LIN {X 0,Y 197.752,Z 444.521,A -85,B 0,C 180,E1 -22110.162,E2 -22110.162} C_VEL
LIN {X 0,Y 204.908,Z 442.853,A -85,B 0,C 180,E1 -22106.718,E2 -22106.718} C_VEL
LIN {X 0,Y 212.782,Z 440.264,A -85,B 0,C 180,E1 -22103.522,E2 -22103.522} C_VEL
LIN {X 0,Y 223.864,Z 435.745,A -85,B 0,C 180,E1 -22099.941,E2 -22099.941} C_VEL
LIN {X 0,Y 233.532,Z 431.085,A -85,B 0,C 180,E1 -22097.381,E2 -22097.381} C_VEL
LIN {X 0,Y 236.072,Z 429.745,A -85,B 0,C 180,E1 -22096.787,E2 -22096.787} C_VEL
LIN {X 0,Y 232.311,Z 432.152,A -85,B 0,C 180,E1 -22095.84,E2 -22095.84} C_VEL
LIN {X 0,Y 218.81,Z 440.079,A -85,B 0,C 180,E1 -22092.416,E2 -22092.416} C_VEL
LIN {X 0,Y 207.624,Z 445.92,A -85,B 0,C 180,E1 -22088.772,E2 -22088.772} C_VEL
LIN {X 0,Y 198.004,Z 450.413,A -85,B 0,C 180,E1 -22084.605,E2 -22084.605} C_VEL
LIN {X 0,Y 191.543,Z 453.093,A -85,B 0,C 180,E1 -22080.909,E2 -22080.909} C_VEL
LIN {X 0,Y 186.17,Z 454.953,A -85,B 0,C 180,E1 -22076.937,E2 -22076.937} C_VEL
LIN {X 0,Y 180.265,Z 456.156,A -85,B 0,C 180,E1 -22070.662,E2 -22070.662} C_VEL
LIN {X 0,Y 178.735,Z 456.196,A -85,B 0,C 180,E1 -22067.89,E2 -22067.89} C_VEL
LIN {X 0,Y 177.023,Z 461.145,A -85,B 0,C 180,E1 -22063.781,E2 -22063.781} C_VEL
LIN {X 0,Y 176.198,Z 465.291,A -85,B 0,C 180,E1 -22059.181,E2 -22059.181} C_VEL
LIN {X 0,Y 175.968,Z 468.104,A -85,B 0,C 180,E1 -22054.582,E2 -22054.582} C_VEL
LIN {X 0,Y 176.016,Z 469.036,A -85,B 0,C 180,E1 -22052.288,E2 -22052.288} C_VEL
LIN {X 0,Y 176.084,Z 469.658,A -85,B 0,C 180,E1 -22050,E2 -22050} C_VEL
LIN {X 0,Y 175.967,Z 469.997,A -85,B 0,C 180,E1 -22045.418,E2 -22045.418} C_VEL
LIN {X 0,Y 176.223,Z 469.176,A -85,B 0,C 180,E1 -22040.821,E2 -22040.821} C_VEL
LIN {X 0,Y 177.152,Z 467.175,A -85,B 0,C 180,E1 -22036.229,E2 -22036.229} C_VEL
LIN {X 0,Y 179.107,Z 463.971,A -85,B 0,C 180,E1 -22031.705,E2 -22031.705} C_VEL
LIN {X 0,Y 182.02,Z 459.529,A -85,B 0,C 180,E1 -22027.287,E2 -22027.287} C_VEL
LIN {X 0,Y 184.225,Z 456.664,A -85,B 0,C 180,E1 -22024.887,E2 -22024.887} C_VEL
LIN {X 0,Y 188.769,Z 455.317,A -85,B 0,C 180,E1 -22021.053,E2 -22021.053} C_VEL
LIN {X 0,Y 198.09,Z 451.582,A -85,B 0,C 180,E1 -22015.413,E2 -22015.413} C_VEL
LIN {X 0,Y 207.59,Z 447.15,A -85,B 0,C 180,E1 -22011.288,E2 -22011.288} C_VEL
LIN {X 0,Y 218.789,Z 441.276,A -85,B 0,C 180,E1 -22007.579,E2 -22007.579} C_VEL
LIN {X 0,Y 231.099,Z 434.128,A -85,B 0,C 180,E1 -22004.383,E2 -22004.383} C_VEL
LIN {X 0,Y 236.096,Z 431.004,A -85,B 0,C 180,E1 -22003.208,E2 -22003.208} C_VEL
LIN {X 0,Y 223.859,Z 436.887,A -85,B 0,C 180,E1 -22000.06,E2 -22000.06} C_VEL
LIN {X 0,Y 216.798,Z 439.813,A -85,B 0,C 180,E1 -21997.857,E2 -21997.857} C_VEL
LIN {X 0,Y 212.822,Z 441.295,A -85,B 0,C 180,E1 -21996.753,E2 -21996.753} C_VEL
LIN {X 0,Y 205.183,Z 443.714,A -85,B 0,C 180,E1 -21995.151,E2 -21995.151} C_VEL
LIN {X 0,Y 197.707,Z 445.563,A -85,B 0,C 180,E1 -21993.403,E2 -21993.403} C_VEL
LIN {X 0,Y 194.059,Z 446.171,A -85,B 0,C 180,E1 -21992.072,E2 -21992.072} C_VEL
LIN {X 0,Y 188.294,Z 446.86,A -85,B 0,C 180,E1 -21989.026,E2 -21989.026} C_VEL
LIN {X 0,Y 182.591,Z 446.752,A -85,B 0,C 180,E1 -21985.048,E2 -21985.048} C_VEL
LIN {X 0,Y 177.835,Z 445.795,A -85,B 0,C 180,E1 -21980.834,E2 -21980.834} C_VEL
LIN {X 0,Y 174.277,Z 443.914,A -85,B 0,C 180,E1 -21976.396,E2 -21976.396} C_VEL
LIN {X 0,Y 171.72,Z 441.035,A -85,B 0,C 180,E1 -21971.807,E2 -21971.807} C_VEL
LIN {X 0,Y 170.045,Z 436.53,A -85,B 0,C 180,E1 -21966.483,E2 -21966.483} C_VEL
LIN {X 0,Y 169.598,Z 432.135,A -85,B 0,C 180,E1 -21962.374,E2 -21962.374} C_VEL
LIN {X 0,Y 169.466,Z 425.713,A -85,B 0,C 180,E1 -21957.622,E2 -21957.622} C_VEL
LIN {X 0,Y 169.738,Z 417.741,A -85,B 0,C 180,E1 -21952.864,E2 -21952.864} C_VEL
LIN {X 0,Y 171.159,Z 419.057,A -85,B 0,C 180,E1 -21950.546,E2 -21950.546} C_VEL
LIN {X 0,Y 178.146,Z 422.179,A -85,B 0,C 180,E1 -21943.968,E2 -21943.968} C_VEL
LIN {X 0,Y 188.053,Z 424.721,A -85,B 0,C 180,E1 -21938.054,E2 -21938.054} C_VEL
LIN {X 0,Y 195.857,Z 426.297,A -85,B 0,C 180,E1 -21934.494,E2 -21934.494} C_VEL
LIN {X 0,Y 190.291,Z 434.455,A -85,B 0,C 180,E1 -21931.305,E2 -21931.305} C_VEL
LIN {X 0,Y 185.284,Z 441.315,A -85,B 0,C 180,E1 -21927.924,E2 -21927.924} C_VEL
LIN {X 0,Y 180.835,Z 447.033,A -85,B 0,C 180,E1 -21924.34,E2 -21924.34} C_VEL
LIN {X 0,Y 177.205,Z 451.661,A -85,B 0,C 180,E1 -21920.611,E2 -21920.611} C_VEL
LIN {X 0,Y 174.129,Z 455.477,A -85,B 0,C 180,E1 -21916.594,E2 -21916.594} C_VEL
LIN {X 0,Y 171.841,Z 458.17,A -85,B 0,C 180,E1 -21912.593,E2 -21912.593} C_VEL
LIN {X 0,Y 170.088,Z 460.1,A -85,B 0,C 180,E1 -21908.271,E2 -21908.271} C_VEL
LIN {X 0,Y 168.834,Z 461.159,A -85,B 0,C 180,E1 -21902.762,E2 -21902.762} C_VEL
LIN {X 0,Y 168.354,Z 460.726,A -85,B 0,C 180,E1 -21897.335,E2 -21897.335} C_VEL
LIN {X 0,Y 168.58,Z 458.874,A -85,B 0,C 180,E1 -21892.037,E2 -21892.037} C_VEL
LIN {X 0,Y 169.593,Z 455.622,A -85,B 0,C 180,E1 -21886.863,E2 -21886.863} C_VEL
LIN {X 0,Y 171.224,Z 450.971,A -85,B 0,C 180,E1 -21881.843,E2 -21881.843} C_VEL
LIN {X 0,Y 173.706,Z 444.826,A -85,B 0,C 180,E1 -21876.972,E2 -21876.972} C_VEL
LIN {X 0,Y 176.584,Z 438.19,A -85,B 0,C 180,E1 -21872.924,E2 -21872.924} C_VEL
LIN {X 0,Y 180.28,Z 429.844,A -85,B 0,C 180,E1 -21868.883,E2 -21868.883} C_VEL
LIN {X 0,Y 184.655,Z 419.915,A -85,B 0,C 180,E1 -21865.087,E2 -21865.087} C_VEL
LIN {X 0,Y 188.981,Z 409.684,A -85,B 0,C 180,E1 -21861.983,E2 -21861.983} C_VEL
LIN {X 0,Y 193.531,Z 397.918,A -85,B 0,C 180,E1 -21859.106,E2 -21859.106} C_VEL
LIN {X 0,Y 198.002,Z 385.301,A -85,B 0,C 180,E1 -21856.661,E2 -21856.661} C_VEL
LIN {X 0,Y 202.09,Z 372.06,A -85,B 0,C 180,E1 -21854.623,E2 -21854.623} C_VEL
LIN {X 0,Y 205.839,Z 357.997,A -85,B 0,C 180,E1 -21852.945,E2 -21852.945} C_VEL
LIN {X 0,Y 208.881,Z 343.591,A -85,B 0,C 180,E1 -21851.613,E2 -21851.613} C_VEL
LIN {X 0,Y 211.287,Z 328.354,A -85,B 0,C 180,E1 -21850.572,E2 -21850.572} C_VEL
LIN {X 0,Y 213.12,Z 312.312,A -85,B 0,C 180,E1 -21849.867,E2 -21849.867} C_VEL
LIN {X 0,Y 219.133,Z 226.935,A -85,B 0,C 180,E1 -21847.267,E2 -21847.267} C_VEL
LIN {X 0,Y 212.064,Z 211.476,A -85,B 0,C 180,E1 -21844.65,E2 -21844.65} C_VEL
LIN {X 0,Y 205.402,Z 198.773,A -85,B 0,C 180,E1 -21842.017,E2 -21842.017} C_VEL
LIN {X 0,Y 198.757,Z 187.359,A -85,B 0,C 180,E1 -21839.182,E2 -21839.182} C_VEL
LIN {X 0,Y 192.968,Z 178.281,A -85,B 0,C 180,E1 -21836.476,E2 -21836.476} C_VEL
LIN {X 0,Y 189.632,Z 173.778,A -85,B 0,C 180,E1 -21834.828,E2 -21834.828} C_VEL
LIN {X 0,Y 186.961,Z 170.012,A -85,B 0,C 180,E1 -21833.413,E2 -21833.413} C_VEL
LIN {X 0,Y 184.1,Z 166.23,A -85,B 0,C 180,E1 -21831.823,E2 -21831.823} C_VEL
LIN {X 0,Y 180.807,Z 162.368,A -85,B 0,C 180,E1 -21829.91,E2 -21829.91} C_VEL
LIN {X 0,Y 179.915,Z 160.782,A -85,B 0,C 180,E1 -21829.317,E2 -21829.317} C_VEL
LIN {X 0,Y 177.199,Z 158.199,A -85,B 0,C 180,E1 -21827.604,E2 -21827.604} C_VEL
LIN {X 0,Y 175.824,Z 158.672,A -85,B 0,C 180,E1 -21826.846,E2 -21826.846} C_VEL
LIN {X 0,Y 174.943,Z 158.617,A -85,B 0,C 180,E1 -21826.271,E2 -21826.271} C_VEL
LIN {X 0,Y 186.878,Z 187.202,A -85,B 0,C 180,E1 -21822.51,E2 -21822.51} C_VEL
LIN {X 0,Y 193.932,Z 204.979,A -85,B 0,C 180,E1 -21820.445,E2 -21820.445} C_VEL
LIN {X 0,Y 185.447,Z 297.749,A -85,B 0,C 180,E1 -21814.479,E2 -21814.479} C_VEL
LIN {X 0,Y 183.681,Z 315.089,A -85,B 0,C 180,E1 -21812.878,E2 -21812.878} C_VEL
LIN {X 0,Y 181.476,Z 332.016,A -85,B 0,C 180,E1 -21810.801,E2 -21810.801} C_VEL
LIN {X 0,Y 179.232,Z 347.562,A -85,B 0,C 180,E1 -21808.389,E2 -21808.389} C_VEL
LIN {X 0,Y 176.911,Z 362.126,A -85,B 0,C 180,E1 -21805.597,E2 -21805.597} C_VEL
LIN {X 0,Y 174.791,Z 375.212,A -85,B 0,C 180,E1 -21802.535,E2 -21802.535} C_VEL
LIN {X 0,Y 172.859,Z 387.807,A -85,B 0,C 180,E1 -21798.982,E2 -21798.982} C_VEL
LIN {X 0,Y 171.565,Z 398.305,A -85,B 0,C 180,E1 -21795.443,E2 -21795.443} C_VEL
LIN {X 0,Y 170.368,Z 408.534,A -85,B 0,C 180,E1 -21791.301,E2 -21791.301} C_VEL
LIN {X 0,Y 169.737,Z 417.09,A -85,B 0,C 180,E1 -21787.136,E2 -21787.136} C_VEL
LIN {X 0,Y 169.426,Z 425.064,A -85,B 0,C 180,E1 -21782.378,E2 -21782.378} C_VEL
LIN {X 0,Y 169.578,Z 431.469,A -85,B 0,C 180,E1 -21777.625,E2 -21777.625} C_VEL
LIN {X 0,Y 170.073,Z 436.447,A -85,B 0,C 180,E1 -21772.879,E2 -21772.879} C_VEL
LIN {X 0,Y 171.659,Z 440.315,A -85,B 0,C 180,E1 -21768.188,E2 -21768.188} C_VEL
LIN {X 0,Y 174.23,Z 443.165,A -85,B 0,C 180,E1 -21763.599,E2 -21763.599} C_VEL
LIN {X 0,Y 177.798,Z 445.006,A -85,B 0,C 180,E1 -21759.161,E2 -21759.161} C_VEL
LIN {X 0,Y 182.543,Z 445.918,A -85,B 0,C 180,E1 -21754.945,E2 -21754.945} C_VEL
LIN {X 0,Y 188.336,Z 445.968,A -85,B 0,C 180,E1 -21750.981,E2 -21750.981} C_VEL
LIN {X 0,Y 195.275,Z 445.044,A -85,B 0,C 180,E1 -21747.327,E2 -21747.327} C_VEL
LIN {X 0,Y 203.134,Z 443.306,A -85,B 0,C 180,E1 -21743.974,E2 -21743.974} C_VEL
LIN {X 0,Y 211.737,Z 440.695,A -85,B 0,C 180,E1 -21740.903,E2 -21740.903} C_VEL
LIN {X 0,Y 223.668,Z 436.148,A -85,B 0,C 180,E1 -21737.503,E2 -21737.503} C_VEL
LIN {X 0,Y 226.162,Z 435.066,A -85,B 0,C 180,E1 -21736.871,E2 -21736.871} C_VEL
LIN {X 0,Y 213.727,Z 441.526,A -85,B 0,C 180,E1 -21733.673,E2 -21733.673} C_VEL
LIN {X 0,Y 204.392,Z 445.882,A -85,B 0,C 180,E1 -21730.792,E2 -21730.792} C_VEL
LIN {X 0,Y 195.993,Z 449.396,A -85,B 0,C 180,E1 -21727.56,E2 -21727.56} C_VEL
LIN {X 0,Y 188.697,Z 452.138,A -85,B 0,C 180,E1 -21723.964,E2 -21723.964} C_VEL
LIN {X 0,Y 182.492,Z 454.047,A -85,B 0,C 180,E1 -21720.043,E2 -21720.043} C_VEL
LIN {X 0,Y 177.444,Z 455.199,A -85,B 0,C 180,E1 -21715.828,E2 -21715.828} C_VEL
LIN {X 0,Y 173.489,Z 455.445,A -85,B 0,C 180,E1 -21711.296,E2 -21711.296} C_VEL
LIN {X 0,Y 172.097,Z 455.258,A -85,B 0,C 180,E1 -21708.914,E2 -21708.914} C_VEL
LIN {X 0,Y 170.076,Z 460.692,A -85,B 0,C 180,E1 -21704.355,E2 -21704.355} C_VEL
LIN {X 0,Y 169.132,Z 464.913,A -85,B 0,C 180,E1 -21699.568,E2 -21699.568} C_VEL
LIN {X 0,Y 168.868,Z 467.797,A -85,B 0,C 180,E1 -21694.775,E2 -21694.775} C_VEL
LIN {X 0,Y 168.925,Z 468.763,A -85,B 0,C 180,E1 -21692.384,E2 -21692.384} C_VEL
LIN {X 0,Y 168.993,Z 469.42,A -85,B 0,C 180,E1 -21690,E2 -21690} C_VEL
LIN {X 0,Y 168.868,Z 469.827,A -85,B 0,C 180,E1 -21685.225,E2 -21685.225} C_VEL
LIN {X 0,Y 169.159,Z 469.065,A -85,B 0,C 180,E1 -21680.434,E2 -21680.434} C_VEL
LIN {X 0,Y 170.202,Z 467.106,A -85,B 0,C 180,E1 -21675.655,E2 -21675.655} C_VEL
LIN {X 0,Y 172.323,Z 463.983,A -85,B 0,C 180,E1 -21670.957,E2 -21670.957} C_VEL
LIN {X 0,Y 175.452,Z 459.633,A -85,B 0,C 180,E1 -21666.386,E2 -21666.386} C_VEL
LIN {X 0,Y 178.084,Z 456.259,A -85,B 0,C 180,E1 -21663.642,E2 -21663.642} C_VEL
LIN {X 0,Y 185.549,Z 454.347,A -85,B 0,C 180,E1 -21657.976,E2 -21657.976} C_VEL
LIN {X 0,Y 192.286,Z 451.988,A -85,B 0,C 180,E1 -21654.211,E2 -21654.211} C_VEL
LIN {X 0,Y 200.091,Z 448.917,A -85,B 0,C 180,E1 -21650.785,E2 -21650.785} C_VEL
LIN {X 0,Y 211.298,Z 443.876,A -85,B 0,C 180,E1 -21647.011,E2 -21647.011} C_VEL
LIN {X 0,Y 226.203,Z 436.278,A -85,B 0,C 180,E1 -21643.119,E2 -21643.119} C_VEL
LIN {X 0,Y 216.351,Z 440.148,A -85,B 0,C 180,E1 -21640.517,E2 -21640.517} C_VEL
LIN {X 0,Y 207.344,Z 443.149,A -85,B 0,C 180,E1 -21637.597,E2 -21637.597} C_VEL
LIN {X 0,Y 199.069,Z 445.269,A -85,B 0,C 180,E1 -21634.393,E2 -21634.393} C_VEL
LIN {X 0,Y 194.059,Z 446.171,A -85,B 0,C 180,E1 -21632.072,E2 -21632.072} C_VEL
LIN {X 0,Y 190.515,Z 446.695,A -85,B 0,C 180,E1 -21630.668,E2 -21630.668} C_VEL
LIN {X 0,Y 183.584,Z 447.267,A -85,B 0,C 180,E1 -21628.503,E2 -21628.503} C_VEL
LIN {X 0,Y 177.068,Z 447.238,A -85,B 0,C 180,E1 -21626.15,E2 -21626.15} C_VEL
LIN {X 0,Y 174.246,Z 446.845,A -85,B 0,C 180,E1 -21624.472,E2 -21624.472} C_VEL
LIN {X 0,Y 169.223,Z 444.931,A -85,B 0,C 180,E1 -21619.405,E2 -21619.405} C_VEL
LIN {X 0,Y 165.985,Z 442.288,A -85,B 0,C 180,E1 -21614.716,E2 -21614.716} C_VEL
LIN {X 0,Y 163.795,Z 438.631,A -85,B 0,C 180,E1 -21609.882,E2 -21609.882} C_VEL
LIN {X 0,Y 162.824,Z 433.883,A -85,B 0,C 180,E1 -21604.952,E2 -21604.952} C_VEL
LIN {X 0,Y 162.479,Z 427.882,A -85,B 0,C 180,E1 -21599.999,E2 -21599.999} C_VEL
LIN {X 0,Y 162.49,Z 421.363,A -85,B 0,C 180,E1 -21595.58,E2 -21595.58} C_VEL
LIN {X 0,Y 162.431,Z 421.883,A -85,B 0,C 180,E1 -21595.035,E2 -21595.035} C_VEL
LIN {X 0,Y 164.208,Z 422.569,A -85,B 0,C 180,E1 -21592.622,E2 -21592.622} C_VEL
LIN {X 0,Y 170.104,Z 425.664,A -85,B 0,C 180,E1 -21585.646,E2 -21585.646} C_VEL
LIN {X 0,Y 179.06,Z 428.214,A -85,B 0,C 180,E1 -21579.313,E2 -21579.313} C_VEL
LIN {X 0,Y 188.158,Z 429.9,A -85,B 0,C 180,E1 -21574.855,E2 -21574.855} C_VEL
LIN {X 0,Y 185.966,Z 433.292,A -85,B 0,C 180,E1 -21573.374,E2 -21573.374} C_VEL
LIN {X 0,Y 179.747,Z 441.34,A -85,B 0,C 180,E1 -21569.449,E2 -21569.449} C_VEL
LIN {X 0,Y 174.113,Z 448.169,A -85,B 0,C 180,E1 -21565.005,E2 -21565.005} C_VEL
LIN {X 0,Y 169.462,Z 453.604,A -85,B 0,C 180,E1 -21560.107,E2 -21560.107} C_VEL
LIN {X 0,Y 166.437,Z 456.96,A -85,B 0,C 180,E1 -21555.877,E2 -21555.877} C_VEL
LIN {X 0,Y 164.876,Z 458.669,A -85,B 0,C 180,E1 -21553.001,E2 -21553.001} C_VEL
LIN {X 0,Y 163.256,Z 460.249,A -85,B 0,C 180,E1 -21549.204,E2 -21549.204} C_VEL
LIN {X 0,Y 161.965,Z 461.303,A -85,B 0,C 180,E1 -21544.34,E2 -21544.34} C_VEL
LIN {X 0,Y 161.33,Z 461.235,A -85,B 0,C 180,E1 -21539.393,E2 -21539.393} C_VEL
LIN {X 0,Y 161.328,Z 459.831,A -85,B 0,C 180,E1 -21533.816,E2 -21533.816} C_VEL
LIN {X 0,Y 161.691,Z 458.188,A -85,B 0,C 180,E1 -21530.348,E2 -21530.348} C_VEL
LIN {X 0,Y 162.605,Z 455.542,A -85,B 0,C 180,E1 -21526.316,E2 -21526.316} C_VEL
LIN {X 0,Y 163.872,Z 452.097,A -85,B 0,C 180,E1 -21522.382,E2 -21522.382} C_VEL
LIN {X 0,Y 166.281,Z 446.218,A -85,B 0,C 180,E1 -21517.285,E2 -21517.285} C_VEL
LIN {X 0,Y 168.957,Z 440.314,A -85,B 0,C 180,E1 -21513.311,E2 -21513.311} C_VEL
LIN {X 0,Y 172.859,Z 431.842,A -85,B 0,C 180,E1 -21508.835,E2 -21508.835} C_VEL
LIN {X 0,Y 177.307,Z 422.259,A -85,B 0,C 180,E1 -21504.883,E2 -21504.883} C_VEL
LIN {X 0,Y 181.69,Z 412.444,A -85,B 0,C 180,E1 -21501.66,E2 -21501.66} C_VEL
LIN {X 0,Y 186.367,Z 401.079,A -85,B 0,C 180,E1 -21498.663,E2 -21498.663} C_VEL
LIN {X 0,Y 190.868,Z 389.142,A -85,B 0,C 180,E1 -21496.153,E2 -21496.153} C_VEL
LIN {X 0,Y 195.053,Z 376.654,A -85,B 0,C 180,E1 -21494.054,E2 -21494.054} C_VEL
LIN {X 0,Y 199.088,Z 362.558,A -85,B 0,C 180,E1 -21492.19,E2 -21492.19} C_VEL
LIN {X 0,Y 202.47,Z 348.304,A -85,B 0,C 180,E1 -21490.746,E2 -21490.746} C_VEL
LIN {X 0,Y 205.199,Z 333.062,A -85,B 0,C 180,E1 -21489.579,E2 -21489.579} C_VEL
LIN {X 0,Y 207.318,Z 317,A -85,B 0,C 180,E1 -21488.758,E2 -21488.758} C_VEL
LIN {X 0,Y 211.081,Z 267.637,A -85,B 0,C 180,E1 -21487.203,E2 -21487.203} C_VEL
LIN {X 0,Y 213.827,Z 229.155,A -85,B 0,C 180,E1 -21486.013,E2 -21486.013} C_VEL
LIN {X 0,Y 206.285,Z 212.672,A -85,B 0,C 180,E1 -21483.049,E2 -21483.049} C_VEL
LIN {X 0,Y 198.503,Z 198.192,A -85,B 0,C 180,E1 -21479.745,E2 -21479.745} C_VEL
LIN {X 0,Y 190.795,Z 185.373,A -85,B 0,C 180,E1 -21476.084,E2 -21476.084} C_VEL
LIN {X 0,Y 186.695,Z 179.623,A -85,B 0,C 180,E1 -21473.987,E2 -21473.987} C_VEL
LIN {X 0,Y 183.777,Z 175.577,A -85,B 0,C 180,E1 -21472.369,E2 -21472.369} C_VEL
LIN {X 0,Y 180.507,Z 171.271,A -85,B 0,C 180,E1 -21470.468,E2 -21470.468} C_VEL
LIN {X 0,Y 177.826,Z 167.753,A -85,B 0,C 180,E1 -21468.777,E2 -21468.777} C_VEL
LIN {X 0,Y 176.593,Z 166.336,A -85,B 0,C 180,E1 -21467.973,E2 -21467.973} C_VEL
LIN {X 0,Y 176.143,Z 166.166,A -85,B 0,C 180,E1 -21467.702,E2 -21467.702} C_VEL
LIN {X 0,Y 174.564,Z 168.912,A -85,B 0,C 180,E1 -21467.028,E2 -21467.028} C_VEL
LIN {X 0,Y 173.507,Z 169.87,A -85,B 0,C 180,E1 -21466.481,E2 -21466.481} C_VEL
LIN {X 0,Y 172.35,Z 169.999,A -85,B 0,C 180,E1 -21465.708,E2 -21465.708} C_VEL
LIN {X 0,Y 184.525,Z 199.879,A -85,B 0,C 180,E1 -21461.834,E2 -21461.834} C_VEL
LIN {X 0,Y 187.026,Z 206.321,A -85,B 0,C 180,E1 -21461.071,E2 -21461.071} C_VEL
LIN {X 0,Y 178.45,Z 297.836,A -85,B 0,C 180,E1 -21454.911,E2 -21454.911} C_VEL
LIN {X 0,Y 176.791,Z 314.188,A -85,B 0,C 180,E1 -21453.358,E2 -21453.358} C_VEL
LIN {X 0,Y 174.824,Z 329.233,A -85,B 0,C 180,E1 -21451.508,E2 -21451.508} C_VEL
LIN {X 0,Y 172.656,Z 343.959,A -85,B 0,C 180,E1 -21449.241,E2 -21449.241} C_VEL
LIN {X 0,Y 170.25,Z 359.1,A -85,B 0,C 180,E1 -21446.345,E2 -21446.345} C_VEL
LIN {X 0,Y 168.077,Z 372.501,A -85,B 0,C 180,E1 -21443.217,E2 -21443.217} C_VEL
LIN {X 0,Y 166.146,Z 384.699,A -85,B 0,C 180,E1 -21439.78,E2 -21439.78} C_VEL
LIN {X 0,Y 164.525,Z 397.347,A -85,B 0,C 180,E1 -21435.486,E2 -21435.486} C_VEL
LIN {X 0,Y 163.33,Z 407.747,A -85,B 0,C 180,E1 -21431.166,E2 -21431.166} C_VEL
LIN {X 0,Y 162.765,Z 415.284,A -85,B 0,C 180,E1 -21427.444,E2 -21427.444} C_VEL
LIN {X 0,Y 162.458,Z 421.776,A -85,B 0,C 180,E1 -21423.721,E2 -21423.721} C_VEL
LIN {X 0,Y 162.455,Z 427.202,A -85,B 0,C 180,E1 -21420.001,E2 -21420.001} C_VEL
LIN {X 0,Y 162.787,Z 433.184,A -85,B 0,C 180,E1 -21415.047,E2 -21415.047} C_VEL
LIN {X 0,Y 163.792,Z 437.913,A -85,B 0,C 180,E1 -21410.118,E2 -21410.118} C_VEL
LIN {X 0,Y 165.933,Z 441.545,A -85,B 0,C 180,E1 -21405.279,E2 -21405.279} C_VEL
LIN {X 0,Y 169.181,Z 444.153,A -85,B 0,C 180,E1 -21400.59,E2 -21400.59} C_VEL
LIN {X 0,Y 173.512,Z 445.883,A -85,B 0,C 180,E1 -21396.107,E2 -21396.107} C_VEL
LIN {X 0,Y 179.001,Z 446.651,A -85,B 0,C 180,E1 -21391.892,E2 -21391.892} C_VEL
LIN {X 0,Y 185.715,Z 446.571,A -85,B 0,C 180,E1 -21388.009,E2 -21388.009} C_VEL
LIN {X 0,Y 193.441,Z 445.606,A -85,B 0,C 180,E1 -21384.459,E2 -21384.459} C_VEL
LIN {X 0,Y 201.914,Z 443.826,A -85,B 0,C 180,E1 -21381.207,E2 -21381.207} C_VEL
LIN {X 0,Y 211.255,Z 441.206,A -85,B 0,C 180,E1 -21378.291,E2 -21378.291} C_VEL
LIN {X 0,Y 216.229,Z 439.515,A -85,B 0,C 180,E1 -21376.957,E2 -21376.957} C_VEL
LIN {X 0,Y 203.811,Z 444.957,A -85,B 0,C 180,E1 -21373.603,E2 -21373.603} C_VEL
LIN {X 0,Y 194.632,Z 448.447,A -85,B 0,C 180,E1 -21370.539,E2 -21370.539} C_VEL
LIN {X 0,Y 186.494,Z 451.22,A -85,B 0,C 180,E1 -21367.082,E2 -21367.082} C_VEL
LIN {X 0,Y 176.346,Z 453.876,A -85,B 0,C 180,E1 -21361.205,E2 -21361.205} C_VEL
LIN {X 0,Y 171.051,Z 454.673,A -85,B 0,C 180,E1 -21356.869,E2 -21356.869} C_VEL
LIN {X 0,Y 165.88,Z 454.47,A -85,B 0,C 180,E1 -21350.612,E2 -21350.612} C_VEL
LIN {X 0,Y 165.427,Z 454.518,A -85,B 0,C 180,E1 -21349.869,E2 -21349.869} C_VEL
LIN {X 0,Y 163.158,Z 460.236,A -85,B 0,C 180,E1 -21344.978,E2 -21344.978} C_VEL
LIN {X 0,Y 162.091,Z 464.532,A -85,B 0,C 180,E1 -21339.988,E2 -21339.988} C_VEL
LIN {X 0,Y 161.765,Z 467.49,A -85,B 0,C 180,E1 -21334.985,E2 -21334.985} C_VEL
LIN {X 0,Y 161.835,Z 468.492,A -85,B 0,C 180,E1 -21332.489,E2 -21332.489} C_VEL
LIN {X 0,Y 161.904,Z 469.183,A -85,B 0,C 180,E1 -21330,E2 -21330} C_VEL
LIN {X 0,Y 161.765,Z 469.656,A -85,B 0,C 180,E1 -21325.015,E2 -21325.015} C_VEL
LIN {X 0,Y 162.119,Z 468.934,A -85,B 0,C 180,E1 -21320.014,E2 -21320.014} C_VEL
LIN {X 0,Y 163.275,Z 467.049,A -85,B 0,C 180,E1 -21315.033,E2 -21315.033} C_VEL
LIN {X 0,Y 165.573,Z 464.005,A -85,B 0,C 180,E1 -21310.149,E2 -21310.149} C_VEL
LIN {X 0,Y 168.922,Z 459.737,A -85,B 0,C 180,E1 -21305.414,E2 -21305.414} C_VEL
LIN {X 0,Y 172.483,Z 455.67,A -85,B 0,C 180,E1 -21301.892,E2 -21301.892} C_VEL
LIN {X 0,Y 179.545,Z 454.278,A -85,B 0,C 180,E1 -21296.769,E2 -21296.769} C_VEL
LIN {X 0,Y 186.571,Z 452.33,A -85,B 0,C 180,E1 -21292.936,E2 -21292.936} C_VEL
LIN {X 0,Y 194.682,Z 449.568,A -85,B 0,C 180,E1 -21289.473,E2 -21289.473} C_VEL
LIN {X 0,Y 206.252,Z 445.084,A -85,B 0,C 180,E1 -21285.691,E2 -21285.691} C_VEL
LIN {X 0,Y 216.213,Z 440.667,A -85,B 0,C 180,E1 -21283.047,E2 -21283.047} C_VEL
LIN {X 0,Y 206.525,Z 443.695,A -85,B 0,C 180,E1 -21280.283,E2 -21280.283} C_VEL
LIN {X 0,Y 197.54,Z 445.826,A -85,B 0,C 180,E1 -21277.215,E2 -21277.215} C_VEL
LIN {X 0,Y 188.196,Z 447.276,A -85,B 0,C 180,E1 -21273.22,E2 -21273.22} C_VEL
LIN {X 0,Y 182.153,Z 447.621,A -85,B 0,C 180,E1 -21270.104,E2 -21270.104} C_VEL
LIN {X 0,Y 174.246,Z 446.845,A -85,B 0,C 180,E1 -21264.472,E2 -21264.472} C_VEL
LIN {X 0,Y 171.588,Z 446.311,A -85,B 0,C 180,E1 -21262.732,E2 -21262.732} C_VEL
LIN {X 0,Y 165.998,Z 444.979,A -85,B 0,C 180,E1 -21259.988,E2 -21259.988} C_VEL
LIN {X 0,Y 161.753,Z 443.51,A -85,B 0,C 180,E1 -21257.698,E2 -21257.698} C_VEL
LIN {X 0,Y 159.486,Z 442.165,A -85,B 0,C 180,E1 -21255.81,E2 -21255.81} C_VEL
LIN {X 0,Y 159.021,Z 441.672,A -85,B 0,C 180,E1 -21255.145,E2 -21255.145} C_VEL
LIN {X 0,Y 156.862,Z 437.881,A -85,B 0,C 180,E1 -21250.323,E2 -21250.323} C_VEL
LIN {X 0,Y 155.826,Z 432.889,A -85,B 0,C 180,E1 -21245.174,E2 -21245.174} C_VEL
LIN {X 0,Y 155.526,Z 428.257,A -85,B 0,C 180,E1 -21241.294,E2 -21241.294} C_VEL
LIN {X 0,Y 155.455,Z 424.927,A -85,B 0,C 180,E1 -21238.704,E2 -21238.704} C_VEL
LIN {X 0,Y 155.517,Z 425.68,A -85,B 0,C 180,E1 -21237.409,E2 -21237.409} C_VEL
LIN {X 0,Y 158.71,Z 427.004,A -85,B 0,C 180,E1 -21232.365,E2 -21232.365} C_VEL
LIN {X 0,Y 164.595,Z 429.866,A -85,B 0,C 180,E1 -21225.155,E2 -21225.155} C_VEL
LIN {X 0,Y 173.614,Z 432.242,A -85,B 0,C 180,E1 -21218.633,E2 -21218.633} C_VEL
LIN {X 0,Y 177.337,Z 432.9,A -85,B 0,C 180,E1 -21216.652,E2 -21216.652} C_VEL
LIN {X 0,Y 180.13,Z 434.366,A -85,B 0,C 180,E1 -21214.584,E2 -21214.584} C_VEL
LIN {X 0,Y 174.38,Z 441.343,A -85,B 0,C 180,E1 -21211.076,E2 -21211.076} C_VEL
LIN {X 0,Y 168.381,Z 448.162,A -85,B 0,C 180,E1 -21206.592,E2 -21206.592} C_VEL
LIN {X 0,Y 163.887,Z 453.049,A -85,B 0,C 180,E1 -21202.187,E2 -21202.187} C_VEL
LIN {X 0,Y 160.607,Z 456.439,A -85,B 0,C 180,E1 -21198.065,E2 -21198.065} C_VEL
LIN {X 0,Y 158.629,Z 458.413,A -85,B 0,C 180,E1 -21194.855,E2 -21194.855} C_VEL
LIN {X 0,Y 156.069,Z 460.723,A -85,B 0,C 180,E1 -21189.083,E2 -21189.083} C_VEL
LIN {X 0,Y 155.072,Z 461.463,A -85,B 0,C 180,E1 -21185.334,E2 -21185.334} C_VEL
LIN {X 0,Y 154.298,Z 461.444,A -85,B 0,C 180,E1 -21180.068,E2 -21180.068} C_VEL
LIN {X 0,Y 154.219,Z 460.093,A -85,B 0,C 180,E1 -21174.214,E2 -21174.214} C_VEL
LIN {X 0,Y 154.928,Z 457.346,A -85,B 0,C 180,E1 -21168.514,E2 -21168.514} C_VEL
LIN {X 0,Y 156.053,Z 454.326,A -85,B 0,C 180,E1 -21164.341,E2 -21164.341} C_VEL
LIN {X 0,Y 158.209,Z 449.087,A -85,B 0,C 180,E1 -21158.945,E2 -21158.945} C_VEL
LIN {X 0,Y 161.244,Z 442.469,A -85,B 0,C 180,E1 -21153.865,E2 -21153.865} C_VEL
LIN {X 0,Y 164.875,Z 434.901,A -85,B 0,C 180,E1 -21149.389,E2 -21149.389} C_VEL
LIN {X 0,Y 169.279,Z 425.922,A -85,B 0,C 180,E1 -21145.237,E2 -21145.237} C_VEL
LIN {X 0,Y 173.595,Z 416.739,A -85,B 0,C 180,E1 -21141.854,E2 -21141.854} C_VEL
LIN {X 0,Y 178.423,Z 405.852,A -85,B 0,C 180,E1 -21138.641,E2 -21138.641} C_VEL
LIN {X 0,Y 183.268,Z 393.94,A -85,B 0,C 180,E1 -21135.849,E2 -21135.849} C_VEL
LIN {X 0,Y 187.987,Z 380.924,A -85,B 0,C 180,E1 -21133.437,E2 -21133.437} C_VEL
LIN {X 0,Y 192.156,Z 367.643,A -85,B 0,C 180,E1 -21131.504,E2 -21131.504} C_VEL
LIN {X 0,Y 195.844,Z 353.695,A -85,B 0,C 180,E1 -21129.931,E2 -21129.931} C_VEL
LIN {X 0,Y 198.715,Z 340.032,A -85,B 0,C 180,E1 -21128.745,E2 -21128.745} C_VEL
LIN {X 0,Y 201.1,Z 325.045,A -85,B 0,C 180,E1 -21127.798,E2 -21127.798} C_VEL
LIN {X 0,Y 202.898,Z 308.513,A -85,B 0,C 180,E1 -21127.134,E2 -21127.134} C_VEL
LIN {X 0,Y 208.623,Z 231.637,A -85,B 0,C 180,E1 -21124.732,E2 -21124.732} C_VEL
LIN {X 0,Y 202.294,Z 217.474,A -85,B 0,C 180,E1 -21122.087,E2 -21122.087} C_VEL
LIN {X 0,Y 194.722,Z 203.09,A -85,B 0,C 180,E1 -21118.713,E2 -21118.713} C_VEL
LIN {X 0,Y 187.484,Z 190.772,A -85,B 0,C 180,E1 -21115.107,E2 -21115.107} C_VEL
LIN {X 0,Y 181.258,Z 181.809,A -85,B 0,C 180,E1 -21111.656,E2 -21111.656} C_VEL
LIN {X 0,Y 178,Z 177.436,A -85,B 0,C 180,E1 -21109.678,E2 -21109.678} C_VEL
LIN {X 0,Y 176.225,Z 175.304,A -85,B 0,C 180,E1 -21108.544,E2 -21108.544} C_VEL
LIN {X 0,Y 175.126,Z 175.501,A -85,B 0,C 180,E1 -21107.944,E2 -21107.944} C_VEL
LIN {X 0,Y 173.898,Z 176.636,A -85,B 0,C 180,E1 -21107.335,E2 -21107.335} C_VEL
LIN {X 0,Y 172.376,Z 179.755,A -85,B 0,C 180,E1 -21106.711,E2 -21106.711} C_VEL
LIN {X 0,Y 170.941,Z 181.31,A -85,B 0,C 180,E1 -21105.993,E2 -21105.993} C_VEL
LIN {X 0,Y 169.593,Z 181.308,A -85,B 0,C 180,E1 -21105.147,E2 -21105.147} C_VEL
LIN {X 0,Y 180.163,Z 207.812,A -85,B 0,C 180,E1 -21101.702,E2 -21101.702} C_VEL
LIN {X 0,Y 171.609,Z 296.917,A -85,B 0,C 180,E1 -21095.434,E2 -21095.434} C_VEL
LIN {X 0,Y 169.733,Z 314.729,A -85,B 0,C 180,E1 -21093.68,E2 -21093.68} C_VEL
LIN {X 0,Y 167.588,Z 330.664,A -85,B 0,C 180,E1 -21091.616,E2 -21091.616} C_VEL
LIN {X 0,Y 165.165,Z 346.746,A -85,B 0,C 180,E1 -21088.949,E2 -21088.949} C_VEL
LIN {X 0,Y 162.753,Z 361.408,A -85,B 0,C 180,E1 -21085.927,E2 -21085.927} C_VEL
LIN {X 0,Y 160.536,Z 374.944,A -85,B 0,C 180,E1 -21082.524,E2 -21082.524} C_VEL
LIN {X 0,Y 158.624,Z 387.351,A -85,B 0,C 180,E1 -21078.738,E2 -21078.738} C_VEL
LIN {X 0,Y 157.085,Z 399.5,A -85,B 0,C 180,E1 -21074.246,E2 -21074.246} C_VEL
LIN {X 0,Y 156.093,Z 409.609,A -85,B 0,C 180,E1 -21069.721,E2 -21069.721} C_VEL
LIN {X 0,Y 155.558,Z 418.023,A -85,B 0,C 180,E1 -21065.185,E2 -21065.185} C_VEL
LIN {X 0,Y 155.453,Z 425.874,A -85,B 0,C 180,E1 -21060.001,E2 -21060.001} C_VEL
LIN {X 0,Y 155.687,Z 430.709,A -85,B 0,C 180,E1 -21056.118,E2 -21056.118} C_VEL
LIN {X 0,Y 156.859,Z 437.145,A -85,B 0,C 180,E1 -21049.677,E2 -21049.677} C_VEL
LIN {X 0,Y 159.102,Z 441.071,A -85,B 0,C 180,E1 -21044.632,E2 -21044.632} C_VEL
LIN {X 0,Y 162.489,Z 444.021,A -85,B 0,C 180,E1 -21039.757,E2 -21039.757} C_VEL
LIN {X 0,Y 167.037,Z 446.004,A -85,B 0,C 180,E1 -21035.119,E2 -21035.119} C_VEL
LIN {X 0,Y 172.784,Z 447.171,A -85,B 0,C 180,E1 -21030.785,E2 -21030.785} C_VEL
LIN {X 0,Y 179.773,Z 447.399,A -85,B 0,C 180,E1 -21026.818,E2 -21026.818} C_VEL
LIN {X 0,Y 187.801,Z 446.826,A -85,B 0,C 180,E1 -21023.22,E2 -21023.22} C_VEL
LIN {X 0,Y 196.574,Z 445.408,A -85,B 0,C 180,E1 -21019.944,E2 -21019.944} C_VEL
LIN {X 0,Y 206.21,Z 443.191,A -85,B 0,C 180,E1 -21017.029,E2 -21017.029} C_VEL
LIN {X 0,Y 193.954,Z 447.567,A -85,B 0,C 180,E1 -21013.51,E2 -21013.51} C_VEL
LIN {X 0,Y 184.988,Z 450.336,A -85,B 0,C 180,E1 -21010.23,E2 -21010.23} C_VEL
LIN {X 0,Y 177.06,Z 452.3,A -85,B 0,C 180,E1 -21006.541,E2 -21006.541} C_VEL
LIN {X 0,Y 170.283,Z 453.571,A -85,B 0,C 180,E1 -21002.449,E2 -21002.449} C_VEL
LIN {X 0,Y 162.397,Z 454.038,A -85,B 0,C 180,E1 -20995.643,E2 -20995.643} C_VEL
LIN {X 0,Y 158.986,Z 453.554,A -85,B 0,C 180,E1 -20991.066,E2 -20991.066} C_VEL
LIN {X 0,Y 156.76,Z 458.499,A -85,B 0,C 180,E1 -20986.943,E2 -20986.943} C_VEL
LIN {X 0,Y 155.247,Z 463.209,A -85,B 0,C 180,E1 -20981.754,E2 -20981.754} C_VEL
LIN {X 0,Y 154.787,Z 465.826,A -85,B 0,C 180,E1 -20977.829,E2 -20977.829} C_VEL
LIN {X 0,Y 154.737,Z 468.216,A -85,B 0,C 180,E1 -20972.603,E2 -20972.603} C_VEL
LIN {X 0,Y 154.804,Z 468.942,A -85,B 0,C 180,E1 -20970,E2 -20970} C_VEL
LIN {X 0,Y 154.687,Z 469.474,A -85,B 0,C 180,E1 -20964.786,E2 -20964.786} C_VEL
LIN {X 0,Y 155.101,Z 468.803,A -85,B 0,C 180,E1 -20959.557,E2 -20959.557} C_VEL
LIN {X 0,Y 156.377,Z 466.993,A -85,B 0,C 180,E1 -20954.356,E2 -20954.356} C_VEL
LIN {X 0,Y 158.856,Z 464.029,A -85,B 0,C 180,E1 -20949.272,E2 -20949.272} C_VEL
LIN {X 0,Y 162.456,Z 459.861,A -85,B 0,C 180,E1 -20944.367,E2 -20944.367} C_VEL
LIN {X 0,Y 166.917,Z 455.063,A -85,B 0,C 180,E1 -20940.174,E2 -20940.174} C_VEL
LIN {X 0,Y 173.63,Z 454.144,A -85,B 0,C 180,E1 -20935.481,E2 -20935.481} C_VEL
LIN {X 0,Y 185.046,Z 451.425,A -85,B 0,C 180,E1 -20929.785,E2 -20929.785} C_VEL
LIN {X 0,Y 193.989,Z 448.664,A -85,B 0,C 180,E1 -20926.5,E2 -20926.5} C_VEL
LIN {X 0,Y 206.214,Z 444.314,A -85,B 0,C 180,E1 -20922.97,E2 -20922.97} C_VEL
LIN {X 0,Y 192.052,Z 447.237,A -85,B 0,C 180,E1 -20918.469,E2 -20918.469} C_VEL
LIN {X 0,Y 183.677,Z 448.16,A -85,B 0,C 180,E1 -20915.025,E2 -20915.025} C_VEL
LIN {X 0,Y 176.073,Z 448.289,A -85,B 0,C 180,E1 -20911.258,E2 -20911.258} C_VEL
LIN {X 0,Y 169.834,Z 447.54,A -85,B 0,C 180,E1 -20907.077,E2 -20907.077} C_VEL
LIN {X 0,Y 164.624,Z 445.926,A -85,B 0,C 180,E1 -20902.595,E2 -20902.595} C_VEL
LIN {X 0,Y 160.722,Z 443.453,A -85,B 0,C 180,E1 -20897.823,E2 -20897.823} C_VEL
LIN {X 0,Y 159.021,Z 441.672,A -85,B 0,C 180,E1 -20895.145,E2 -20895.145} C_VEL
LIN {X 0,Y 157.367,Z 440.139,A -85,B 0,C 180,E1 -20893.182,E2 -20893.182} C_VEL
LIN {X 0,Y 153.349,Z 437.039,A -85,B 0,C 180,E1 -20890.054,E2 -20890.054} C_VEL
LIN {X 0,Y 149.739,Z 433.363,A -85,B 0,C 180,E1 -20886.826,E2 -20886.826} C_VEL
LIN {X 0,Y 148.79,Z 430.958,A -85,B 0,C 180,E1 -20884.759,E2 -20884.759} C_VEL
LIN {X 0,Y 148.586,Z 428.509,A -85,B 0,C 180,E1 -20882.541,E2 -20882.541} C_VEL
LIN {X 0,Y 148.465,Z 429.045,A -85,B 0,C 180,E1 -20881.355,E2 -20881.355} C_VEL
LIN {X 0,Y 153.04,Z 431.208,A -85,B 0,C 180,E1 -20872.08,E2 -20872.08} C_VEL
LIN {X 0,Y 158.939,Z 433.855,A -85,B 0,C 180,E1 -20864.614,E2 -20864.614} C_VEL
LIN {X 0,Y 171.792,Z 436.673,A -85,B 0,C 180,E1 -20855.851,E2 -20855.851} C_VEL
LIN {X 0,Y 172.587,Z 437.074,A -85,B 0,C 180,E1 -20855.223,E2 -20855.223} C_VEL
LIN {X 0,Y 171.574,Z 438.663,A -85,B 0,C 180,E1 -20854.312,E2 -20854.312} C_VEL
LIN {X 0,Y 165.646,Z 445.212,A -85,B 0,C 180,E1 -20850.432,E2 -20850.432} C_VEL
LIN {X 0,Y 160.498,Z 450.502,A -85,B 0,C 180,E1 -20846.303,E2 -20846.303} C_VEL
LIN {X 0,Y 156.291,Z 454.696,A -85,B 0,C 180,E1 -20841.935,E2 -20841.935} C_VEL
LIN {X 0,Y 152.109,Z 458.556,A -85,B 0,C 180,E1 -20836.126,E2 -20836.126} C_VEL
LIN {X 0,Y 149.676,Z 460.615,A -85,B 0,C 180,E1 -20831.099,E2 -20831.099} C_VEL
LIN {X 0,Y 147.82,Z 461.727,A -85,B 0,C 180,E1 -20824.787,E2 -20824.787} C_VEL
LIN {X 0,Y 147.239,Z 461.652,A -85,B 0,C 180,E1 -20820.774,E2 -20820.774} C_VEL
LIN {X 0,Y 147.079,Z 460.395,A -85,B 0,C 180,E1 -20814.781,E2 -20814.781} C_VEL
LIN {X 0,Y 147.902,Z 457.36,A -85,B 0,C 180,E1 -20808.125,E2 -20808.125} C_VEL
LIN {X 0,Y 149.131,Z 454.17,A -85,B 0,C 180,E1 -20803.629,E2 -20803.629} C_VEL
LIN {X 0,Y 151.452,Z 448.824,A -85,B 0,C 180,E1 -20798.002,E2 -20798.002} C_VEL
LIN {X 0,Y 154.821,Z 441.911,A -85,B 0,C 180,E1 -20792.602,E2 -20792.602} C_VEL
LIN {X 0,Y 158.63,Z 434.381,A -85,B 0,C 180,E1 -20788.096,E2 -20788.096} C_VEL
LIN {X 0,Y 162.703,Z 426.449,A -85,B 0,C 180,E1 -20784.338,E2 -20784.338} C_VEL
LIN {X 0,Y 167.885,Z 415.899,A -85,B 0,C 180,E1 -20780.361,E2 -20780.361} C_VEL
LIN {X 0,Y 173.088,Z 404.595,A -85,B 0,C 180,E1 -20777.033,E2 -20777.033} C_VEL
LIN {X 0,Y 178.054,Z 392.659,A -85,B 0,C 180,E1 -20774.254,E2 -20774.254} C_VEL
LIN {X 0,Y 183.002,Z 379.334,A -85,B 0,C 180,E1 -20771.818,E2 -20771.818} C_VEL
LIN {X 0,Y 187.558,Z 364.843,A -85,B 0,C 180,E1 -20769.77,E2 -20769.77} C_VEL
LIN {X 0,Y 191.138,Z 351.147,A -85,B 0,C 180,E1 -20768.285,E2 -20768.285} C_VEL
LIN {X 0,Y 194.214,Z 335.891,A -85,B 0,C 180,E1 -20767.037,E2 -20767.037} C_VEL
LIN {X 0,Y 196.459,Z 321.055,A -85,B 0,C 180,E1 -20766.199,E2 -20766.199} C_VEL
LIN {X 0,Y 198.373,Z 300.438,A -85,B 0,C 180,E1 -20765.47,E2 -20765.47} C_VEL
LIN {X 0,Y 203.602,Z 234.224,A -85,B 0,C 180,E1 -20763.417,E2 -20763.417} C_VEL
LIN {X 0,Y 197.616,Z 220.8,A -85,B 0,C 180,E1 -20760.78,E2 -20760.78} C_VEL
LIN {X 0,Y 190.735,Z 207.401,A -85,B 0,C 180,E1 -20757.5,E2 -20757.5} C_VEL
LIN {X 0,Y 183.99,Z 195.794,A -85,B 0,C 180,E1 -20753.962,E2 -20753.962} C_VEL
LIN {X 0,Y 178.302,Z 187.516,A -85,B 0,C 180,E1 -20750.651,E2 -20750.651} C_VEL
LIN {X 0,Y 176.163,Z 184.475,A -85,B 0,C 180,E1 -20749.29,E2 -20749.29} C_VEL
LIN {X 0,Y 174.531,Z 184.339,A -85,B 0,C 180,E1 -20748.382,E2 -20748.382} C_VEL
LIN {X 0,Y 172.335,Z 187.119,A -85,B 0,C 180,E1 -20747.363,E2 -20747.363} C_VEL
LIN {X 0,Y 171.227,Z 187.998,A -85,B 0,C 180,E1 -20746.783,E2 -20746.783} C_VEL
LIN {X 0,Y 169.55,Z 191.433,A -85,B 0,C 180,E1 -20746.09,E2 -20746.09} C_VEL
LIN {X 0,Y 168.067,Z 192.983,A -85,B 0,C 180,E1 -20745.308,E2 -20745.308} C_VEL
LIN {X 0,Y 166.945,Z 192.992,A -85,B 0,C 180,E1 -20744.576,E2 -20744.576} C_VEL
LIN {X 0,Y 173.29,Z 209.163,A -85,B 0,C 180,E1 -20742.379,E2 -20742.379} C_VEL
LIN {X 0,Y 164.518,Z 297.928,A -85,B 0,C 180,E1 -20735.813,E2 -20735.813} C_VEL
LIN {X 0,Y 162.615,Z 315.349,A -85,B 0,C 180,E1 -20733.997,E2 -20733.997} C_VEL
LIN {X 0,Y 160.357,Z 331.822,A -85,B 0,C 180,E1 -20731.732,E2 -20731.732} C_VEL
LIN {X 0,Y 157.908,Z 347.73,A -85,B 0,C 180,E1 -20728.949,E2 -20728.949} C_VEL
LIN {X 0,Y 155.399,Z 362.588,A -85,B 0,C 180,E1 -20725.697,E2 -20725.697} C_VEL
LIN {X 0,Y 153.082,Z 376.706,A -85,B 0,C 180,E1 -20721.9,E2 -20721.9} C_VEL
LIN {X 0,Y 151.098,Z 389.752,A -85,B 0,C 180,E1 -20717.599,E2 -20717.599} C_VEL
LIN {X 0,Y 150.087,Z 398.42,A -85,B 0,C 180,E1 -20714.232,E2 -20714.232} C_VEL
LIN {X 0,Y 149.086,Z 408.689,A -85,B 0,C 180,E1 -20709.498,E2 -20709.498} C_VEL
LIN {X 0,Y 148.591,Z 417.234,A -85,B 0,C 180,E1 -20704.749,E2 -20704.749} C_VEL
LIN {X 0,Y 148.492,Z 424.349,A -85,B 0,C 180,E1 -20700.001,E2 -20700.001} C_VEL
LIN {X 0,Y 148.733,Z 429.452,A -85,B 0,C 180,E1 -20695.936,E2 -20695.936} C_VEL
LIN {X 0,Y 149.942,Z 436.28,A -85,B 0,C 180,E1 -20689.195,E2 -20689.195} C_VEL
LIN {X 0,Y 152.3,Z 440.485,A -85,B 0,C 180,E1 -20683.927,E2 -20683.927} C_VEL
LIN {X 0,Y 155.843,Z 443.705,A -85,B 0,C 180,E1 -20678.853,E2 -20678.853} C_VEL
LIN {X 0,Y 160.616,Z 446.046,A -85,B 0,C 180,E1 -20674.052,E2 -20674.052} C_VEL
LIN {X 0,Y 166.626,Z 447.485,A -85,B 0,C 180,E1 -20669.594,E2 -20669.594} C_VEL
LIN {X 0,Y 173.906,Z 448.13,A -85,B 0,C 180,E1 -20665.545,E2 -20665.545} C_VEL
LIN {X 0,Y 182.225,Z 447.875,A -85,B 0,C 180,E1 -20661.897,E2 -20661.897} C_VEL
LIN {X 0,Y 193.718,Z 446.493,A -85,B 0,C 180,E1 -20657.843,E2 -20657.843} C_VEL
LIN {X 0,Y 196.168,Z 446.067,A -85,B 0,C 180,E1 -20657.102,E2 -20657.102} C_VEL
LIN {X 0,Y 184.125,Z 449.501,A -85,B 0,C 180,E1 -20653.397,E2 -20653.397} C_VEL
LIN {X 0,Y 171.392,Z 452.226,A -85,B 0,C 180,E1 -20647.958,E2 -20647.958} C_VEL
LIN {X 0,Y 164.314,Z 453.115,A -85,B 0,C 180,E1 -20643.782,E2 -20643.782} C_VEL
LIN {X 0,Y 158.487,Z 453.327,A -85,B 0,C 180,E1 -20639.195,E2 -20639.195} C_VEL
LIN {X 0,Y 152.64,Z 452.464,A -85,B 0,C 180,E1 -20632.436,E2 -20632.436} C_VEL
LIN {X 0,Y 149.919,Z 457.969,A -85,B 0,C 180,E1 -20627.741,E2 -20627.741} C_VEL
LIN {X 0,Y 148.233,Z 462.764,A -85,B 0,C 180,E1 -20622.319,E2 -20622.319} C_VEL
LIN {X 0,Y 147.723,Z 465.465,A -85,B 0,C 180,E1 -20618.206,E2 -20618.206} C_VEL
LIN {X 0,Y 147.64,Z 467.935,A -85,B 0,C 180,E1 -20612.728,E2 -20612.728} C_VEL
LIN {X 0,Y 147.628,Z 468.918,A -85,B 0,C 180,E1 -20608.637,E2 -20608.637} C_VEL
LIN {X 0,Y 147.607,Z 469.269,A -85,B 0,C 180,E1 -20604.536,E2 -20604.536} C_VEL
LIN {X 0,Y 148.071,Z 468.671,A -85,B 0,C 180,E1 -20599.056,E2 -20599.056} C_VEL
LIN {X 0,Y 149.509,Z 466.944,A -85,B 0,C 180,E1 -20593.618,E2 -20593.618} C_VEL
LIN {X 0,Y 152.184,Z 464.074,A -85,B 0,C 180,E1 -20588.318,E2 -20588.318} C_VEL
LIN {X 0,Y 156.067,Z 459.997,A -85,B 0,C 180,E1 -20583.236,E2 -20583.236} C_VEL
LIN {X 0,Y 161.697,Z 454.424,A -85,B 0,C 180,E1 -20578.197,E2 -20578.197} C_VEL
LIN {X 0,Y 171.476,Z 453.295,A -85,B 0,C 180,E1 -20572.064,E2 -20572.064} C_VEL
LIN {X 0,Y 184.164,Z 450.567,A -85,B 0,C 180,E1 -20566.614,E2 -20566.614} C_VEL
LIN {X 0,Y 196.217,Z 447.117,A -85,B 0,C 180,E1 -20562.884,E2 -20562.884} C_VEL
LIN {X 0,Y 186.634,Z 448.501,A -85,B 0,C 180,E1 -20559.803,E2 -20559.803} C_VEL
LIN {X 0,Y 173.844,Z 449.06,A -85,B 0,C 180,E1 -20554.469,E2 -20554.469} C_VEL
LIN {X 0,Y 166.658,Z 448.364,A -85,B 0,C 180,E1 -20550.4,E2 -20550.4} C_VEL
LIN {X 0,Y 160.676,Z 446.889,A -85,B 0,C 180,E1 -20545.937,E2 -20545.937} C_VEL
LIN {X 0,Y 155.928,Z 444.514,A -85,B 0,C 180,E1 -20541.135,E2 -20541.135} C_VEL
LIN {X 0,Y 152.144,Z 441.003,A -85,B 0,C 180,E1 -20535.732,E2 -20535.732} C_VEL
LIN {X 0,Y 149.946,Z 437.028,A -85,B 0,C 180,E1 -20530.805,E2 -20530.805} C_VEL
LIN {X 0,Y 148.79,Z 430.958,A -85,B 0,C 180,E1 -20524.759,E2 -20524.759} C_VEL
LIN {X 0,Y 148.288,Z 430.248,A -85,B 0,C 180,E1 -20523.551,E2 -20523.551} C_VEL
LIN {X 0,Y 146.869,Z 430.643,A -85,B 0,C 180,E1 -20521.835,E2 -20521.835} C_VEL
LIN {X 0,Y 144.226,Z 433.415,A -85,B 0,C 180,E1 -20518.322,E2 -20518.322} C_VEL
LIN {X 0,Y 144.302,Z 434.141,A -85,B 0,C 180,E1 -20516.712,E2 -20516.712} C_VEL
LIN {X 0,Y 147.198,Z 435.181,A -85,B 0,C 180,E1 -20511.764,E2 -20511.764} C_VEL
LIN {X 0,Y 154.519,Z 437.989,A -85,B 0,C 180,E1 -20502.774,E2 -20502.774} C_VEL
LIN {X 0,Y 165.214,Z 440.059,A -85,B 0,C 180,E1 -20495.495,E2 -20495.495} C_VEL
LIN {X 0,Y 160.604,Z 445.045,A -85,B 0,C 180,E1 -20492.392,E2 -20492.392} C_VEL
LIN {X 0,Y 154.433,Z 451.003,A -85,B 0,C 180,E1 -20487.667,E2 -20487.667} C_VEL
LIN {X 0,Y 149.105,Z 455.843,A -85,B 0,C 180,E1 -20482.21,E2 -20482.21} C_VEL
LIN {X 0,Y 145.123,Z 459.16,A -85,B 0,C 180,E1 -20476.587,E2 -20476.587} C_VEL
LIN {X 0,Y 143.09,Z 460.711,A -85,B 0,C 180,E1 -20472.544,E2 -20472.544} C_VEL
LIN {X 0,Y 141.135,Z 461.871,A -85,B 0,C 180,E1 -20466.695,E2 -20466.695} C_VEL
LIN {X 0,Y 140.08,Z 461.724,A -85,B 0,C 180,E1 -20460.113,E2 -20460.113} C_VEL
LIN {X 0,Y 140.038,Z 460.14,A -85,B 0,C 180,E1 -20453.671,E2 -20453.671} C_VEL
LIN {X 0,Y 140.936,Z 457.163,A -85,B 0,C 180,E1 -20447.41,E2 -20447.41} C_VEL
LIN {X 0,Y 142.252,Z 454.008,A -85,B 0,C 180,E1 -20442.846,E2 -20442.846} C_VEL
LIN {X 0,Y 144.048,Z 450.042,A -85,B 0,C 180,E1 -20438.417,E2 -20438.417} C_VEL
LIN {X 0,Y 147.416,Z 443.39,A -85,B 0,C 180,E1 -20432.733,E2 -20432.733} C_VEL
LIN {X 0,Y 151.231,Z 436.155,A -85,B 0,C 180,E1 -20428.003,E2 -20428.003} C_VEL
LIN {X 0,Y 155.488,Z 428.262,A -85,B 0,C 180,E1 -20423.939,E2 -20423.939} C_VEL
LIN {X 0,Y 160.6,Z 418.369,A -85,B 0,C 180,E1 -20419.919,E2 -20419.919} C_VEL
LIN {X 0,Y 165.628,Z 408.089,A -85,B 0,C 180,E1 -20416.626,E2 -20416.626} C_VEL
LIN {X 0,Y 170.984,Z 396.066,A -85,B 0,C 180,E1 -20413.585,E2 -20413.585} C_VEL
LIN {X 0,Y 176.018,Z 383.394,A -85,B 0,C 180,E1 -20411.07,E2 -20411.07} C_VEL
LIN {X 0,Y 180.789,Z 369.426,A -85,B 0,C 180,E1 -20408.906,E2 -20408.906} C_VEL
LIN {X 0,Y 184.947,Z 355.076,A -85,B 0,C 180,E1 -20407.224,E2 -20407.224} C_VEL
LIN {X 0,Y 188.27,Z 340.328,A -85,B 0,C 180,E1 -20405.903,E2 -20405.903} C_VEL
LIN {X 0,Y 190.822,Z 325.286,A -85,B 0,C 180,E1 -20404.941,E2 -20404.941} C_VEL
LIN {X 0,Y 192.742,Z 308.629,A -85,B 0,C 180,E1 -20404.269,E2 -20404.269} C_VEL
LIN {X 0,Y 198.559,Z 236.515,A -85,B 0,C 180,E1 -20401.991,E2 -20401.991} C_VEL
LIN {X 0,Y 193.402,Z 224.931,A -85,B 0,C 180,E1 -20399.588,E2 -20399.588} C_VEL
LIN {X 0,Y 187.223,Z 212.576,A -85,B 0,C 180,E1 -20396.483,E2 -20396.483} C_VEL
LIN {X 0,Y 180.595,Z 200.851,A -85,B 0,C 180,E1 -20392.786,E2 -20392.786} C_VEL
LIN {X 0,Y 175.278,Z 193.033,A -85,B 0,C 180,E1 -20389.535,E2 -20389.535} C_VEL
LIN {X 0,Y 174.659,Z 192.189,A -85,B 0,C 180,E1 -20389.129,E2 -20389.129} C_VEL
LIN {X 0,Y 172.951,Z 193.616,A -85,B 0,C 180,E1 -20388.303,E2 -20388.303} C_VEL
LIN {X 0,Y 170.904,Z 197.162,A -85,B 0,C 180,E1 -20387.429,E2 -20387.429} C_VEL
LIN {X 0,Y 168.706,Z 199.411,A -85,B 0,C 180,E1 -20386.323,E2 -20386.323} C_VEL
LIN {X 0,Y 168.355,Z 199.904,A -85,B 0,C 180,E1 -20386.154,E2 -20386.154} C_VEL
LIN {X 0,Y 166.695,Z 203.328,A -85,B 0,C 180,E1 -20385.439,E2 -20385.439} C_VEL
LIN {X 0,Y 165.257,Z 204.837,A -85,B 0,C 180,E1 -20384.647,E2 -20384.647} C_VEL
LIN {X 0,Y 164.118,Z 204.744,A -85,B 0,C 180,E1 -20383.858,E2 -20383.858} C_VEL
LIN {X 0,Y 166.441,Z 210.591,A -85,B 0,C 180,E1 -20383.063,E2 -20383.063} C_VEL
LIN {X 0,Y 157.558,Z 297.67,A -85,B 0,C 180,E1 -20376.304,E2 -20376.304} C_VEL
LIN {X 0,Y 155.741,Z 314.138,A -85,B 0,C 180,E1 -20374.535,E2 -20374.535} C_VEL
LIN {X 0,Y 153.421,Z 330.848,A -85,B 0,C 180,E1 -20372.177,E2 -20372.177} C_VEL
LIN {X 0,Y 150.931,Z 346.861,A -85,B 0,C 180,E1 -20369.271,E2 -20369.271} C_VEL
LIN {X 0,Y 148.302,Z 362.225,A -85,B 0,C 180,E1 -20365.788,E2 -20365.788} C_VEL
LIN {X 0,Y 145.999,Z 376.141,A -85,B 0,C 180,E1 -20361.906,E2 -20361.906} C_VEL
LIN {X 0,Y 144.131,Z 388.398,A -85,B 0,C 180,E1 -20357.745,E2 -20357.745} C_VEL
LIN {X 0,Y 142.884,Z 398.765,A -85,B 0,C 180,E1 -20353.512,E2 -20353.512} C_VEL
LIN {X 0,Y 142.004,Z 409.012,A -85,B 0,C 180,E1 -20348.539,E2 -20348.539} C_VEL
LIN {X 0,Y 141.584,Z 417.509,A -85,B 0,C 180,E1 -20343.558,E2 -20343.558} C_VEL
LIN {X 0,Y 141.622,Z 424.548,A -85,B 0,C 180,E1 -20338.579,E2 -20338.579} C_VEL
LIN {X 0,Y 141.922,Z 429.642,A -85,B 0,C 180,E1 -20334.317,E2 -20334.317} C_VEL
LIN {X 0,Y 143.564,Z 436.472,A -85,B 0,C 180,E1 -20327.275,E2 -20327.275} C_VEL
LIN {X 0,Y 147.269,Z 441.65,A -85,B 0,C 180,E1 -20320.486,E2 -20320.486} C_VEL
LIN {X 0,Y 151.591,Z 444.687,A -85,B 0,C 180,E1 -20315.339,E2 -20315.339} C_VEL
LIN {X 0,Y 157.264,Z 446.93,A -85,B 0,C 180,E1 -20310.556,E2 -20310.556} C_VEL
LIN {X 0,Y 164.174,Z 448.273,A -85,B 0,C 180,E1 -20306.186,E2 -20306.186} C_VEL
LIN {X 0,Y 172.28,Z 448.862,A -85,B 0,C 180,E1 -20302.273,E2 -20302.273} C_VEL
LIN {X 0,Y 186.155,Z 448.168,A -85,B 0,C 180,E1 -20297.191,E2 -20297.191} C_VEL
LIN {X 0,Y 174.394,Z 450.653,A -85,B 0,C 180,E1 -20293.243,E2 -20293.243} C_VEL
LIN {X 0,Y 165.842,Z 451.945,A -85,B 0,C 180,E1 -20289.469,E2 -20289.469} C_VEL
LIN {X 0,Y 158.447,Z 452.564,A -85,B 0,C 180,E1 -20285.213,E2 -20285.213} C_VEL
LIN {X 0,Y 149.732,Z 452.107,A -85,B 0,C 180,E1 -20277.993,E2 -20277.993} C_VEL
LIN {X 0,Y 146.45,Z 451.255,A -85,B 0,C 180,E1 -20273.933,E2 -20273.933} C_VEL
LIN {X 0,Y 143.114,Z 457.439,A -85,B 0,C 180,E1 -20268.615,E2 -20268.615} C_VEL
LIN {X 0,Y 141.244,Z 462.32,A -85,B 0,C 180,E1 -20262.939,E2 -20262.939} C_VEL
LIN {X 0,Y 140.654,Z 465.104,A -85,B 0,C 180,E1 -20258.621,E2 -20258.621} C_VEL
LIN {X 0,Y 140.543,Z 467.645,A -85,B 0,C 180,E1 -20252.866,E2 -20252.866} C_VEL
LIN {X 0,Y 140.567,Z 468.554,A -85,B 0,C 180,E1 -20249.354,E2 -20249.354} C_VEL
LIN {X 0,Y 140.524,Z 469.062,A -85,B 0,C 180,E1 -20244.259,E2 -20244.259} C_VEL
LIN {X 0,Y 141.063,Z 468.545,A -85,B 0,C 180,E1 -20238.505,E2 -20238.505} C_VEL
LIN {X 0,Y 142.672,Z 466.903,A -85,B 0,C 180,E1 -20232.809,E2 -20232.809} C_VEL
LIN {X 0,Y 145.542,Z 464.12,A -85,B 0,C 180,E1 -20227.275,E2 -20227.275} C_VEL
LIN {X 0,Y 149.731,Z 460.138,A -85,B 0,C 180,E1 -20222.006,E2 -20222.006} C_VEL
LIN {X 0,Y 155.297,Z 454.848,A -85,B 0,C 180,E1 -20217.107,E2 -20217.107} C_VEL
LIN {X 0,Y 156.695,Z 453.654,A -85,B 0,C 180,E1 -20216.093,E2 -20216.093} C_VEL
LIN {X 0,Y 165.92,Z 452.997,A -85,B 0,C 180,E1 -20210.553,E2 -20210.553} C_VEL
LIN {X 0,Y 174.445,Z 451.69,A -85,B 0,C 180,E1 -20206.773,E2 -20206.773} C_VEL
LIN {X 0,Y 186.178,Z 449.21,A -85,B 0,C 180,E1 -20202.802,E2 -20202.802} C_VEL
LIN {X 0,Y 176.664,Z 449.8,A -85,B 0,C 180,E1 -20199.531,E2 -20199.531} C_VEL
LIN {X 0,Y 168.064,Z 449.596,A -85,B 0,C 180,E1 -20195.834,E2 -20195.834} C_VEL
LIN {X 0,Y 160.575,Z 448.59,A -85,B 0,C 180,E1 -20191.682,E2 -20191.682} C_VEL
LIN {X 0,Y 154.316,Z 446.757,A -85,B 0,C 180,E1 -20187.092,E2 -20187.092} C_VEL
LIN {X 0,Y 149.348,Z 444.099,A -85,B 0,C 180,E1 -20182.114,E2 -20182.114} C_VEL
LIN {X 0,Y 144.814,Z 439.5,A -85,B 0,C 180,E1 -20175.48,E2 -20175.48} C_VEL
LIN {X 0,Y 142.517,Z 434.316,A -85,B 0,C 180,E1 -20169.505,E2 -20169.505} C_VEL
LIN {X 0,Y 142.08,Z 432.17,A -85,B 0,C 180,E1 -20167.235,E2 -20167.235} C_VEL
LIN {X 0,Y 141.839,Z 432.63,A -85,B 0,C 180,E1 -20165.686,E2 -20165.686} C_VEL
LIN {X 0,Y 142.632,Z 432.811,A -85,B 0,C 180,E1 -20162.823,E2 -20162.823} C_VEL
LIN {X 0,Y 144.302,Z 434.141,A -85,B 0,C 180,E1 -20156.712,E2 -20156.712} C_VEL
LIN {X 0,Y 144.849,Z 435.031,A -85,B 0,C 180,E1 -20154.406,E2 -20154.406} C_VEL
LIN {X 0,Y 144.556,Z 437.496,A -85,B 0,C 180,E1 -20150.597,E2 -20150.597} C_VEL
LIN {X 0,Y 144.78,Z 439.947,A -85,B 0,C 180,E1 -20146.776,E2 -20146.776} C_VEL
LIN {X 0,Y 146.135,Z 440.827,A -85,B 0,C 180,E1 -20144.532,E2 -20144.532} C_VEL
LIN {X 0,Y 156.662,Z 443.013,A -85,B 0,C 180,E1 -20136.186,E2 -20136.186} C_VEL
LIN {X 0,Y 155.757,Z 444.888,A -85,B 0,C 180,E1 -20134.48,E2 -20134.48} C_VEL
LIN {X 0,Y 149.779,Z 450.319,A -85,B 0,C 180,E1 -20130.235,E2 -20130.235} C_VEL
LIN {X 0,Y 144.725,Z 454.666,A -85,B 0,C 180,E1 -20125.643,E2 -20125.643} C_VEL
LIN {X 0,Y 141.86,Z 456.954,A -85,B 0,C 180,E1 -20122.436,E2 -20122.436} C_VEL
LIN {X 0,Y 139.381,Z 458.845,A -85,B 0,C 180,E1 -20119.041,E2 -20119.041} C_VEL
LIN {X 0,Y 135.79,Z 461.269,A -85,B 0,C 180,E1 -20112.286,E2 -20112.286} C_VEL
LIN {X 0,Y 134.431,Z 461.968,A -85,B 0,C 180,E1 -20108.352,E2 -20108.352} C_VEL
LIN {X 0,Y 133.146,Z 462.029,A -85,B 0,C 180,E1 -20101.86,E2 -20101.86} C_VEL
LIN {X 0,Y 132.836,Z 460.934,A -85,B 0,C 180,E1 -20095.915,E2 -20095.915} C_VEL
LIN {X 0,Y 133.066,Z 459.507,A -85,B 0,C 180,E1 -20091.698,E2 -20091.698} C_VEL
LIN {X 0,Y 133.604,Z 457.963,A -85,B 0,C 180,E1 -20088.398,E2 -20088.398} C_VEL
LIN {X 0,Y 134.856,Z 454.961,A -85,B 0,C 180,E1 -20083.563,E2 -20083.563} C_VEL
LIN {X 0,Y 137.335,Z 449.74,A -85,B 0,C 180,E1 -20077.35,E2 -20077.35} C_VEL
LIN {X 0,Y 140.639,Z 443.563,A -85,B 0,C 180,E1 -20071.892,E2 -20071.892} C_VEL
LIN {X 0,Y 145.074,Z 435.582,A -85,B 0,C 180,E1 -20066.528,E2 -20066.528} C_VEL
LIN {X 0,Y 150.136,Z 426.615,A -85,B 0,C 180,E1 -20061.927,E2 -20061.927} C_VEL
LIN {X 0,Y 155.04,Z 417.453,A -85,B 0,C 180,E1 -20058.23,E2 -20058.23} C_VEL
LIN {X 0,Y 160.529,Z 406.572,A -85,B 0,C 180,E1 -20054.771,E2 -20054.771} C_VEL
LIN {X 0,Y 165.971,Z 394.676,A -85,B 0,C 180,E1 -20051.803,E2 -20051.803} C_VEL
LIN {X 0,Y 171.249,Z 381.676,A -85,B 0,C 180,E1 -20049.27,E2 -20049.27} C_VEL
LIN {X 0,Y 175.949,Z 368.186,A -85,B 0,C 180,E1 -20047.226,E2 -20047.226} C_VEL
LIN {X 0,Y 179.934,Z 354.531,A -85,B 0,C 180,E1 -20045.634,E2 -20045.634} C_VEL
LIN {X 0,Y 183.366,Z 339.567,A -85,B 0,C 180,E1 -20044.305,E2 -20044.305} C_VEL
LIN {X 0,Y 186.015,Z 324.12,A -85,B 0,C 180,E1 -20043.342,E2 -20043.342} C_VEL
LIN {X 0,Y 187.904,Z 307.629,A -85,B 0,C 180,E1 -20042.706,E2 -20042.706} C_VEL
LIN {X 0,Y 193.666,Z 239.331,A -85,B 0,C 180,E1 -20040.553,E2 -20040.553} C_VEL
LIN {X 0,Y 189.584,Z 229.664,A -85,B 0,C 180,E1 -20038.5,E2 -20038.5} C_VEL
LIN {X 0,Y 183.606,Z 217.488,A -85,B 0,C 180,E1 -20035.34,E2 -20035.34} C_VEL
LIN {X 0,Y 177.69,Z 206.626,A -85,B 0,C 180,E1 -20031.856,E2 -20031.856} C_VEL
LIN {X 0,Y 173.87,Z 200.762,A -85,B 0,C 180,E1 -20029.43,E2 -20029.43} C_VEL
LIN {X 0,Y 170.819,Z 204.607,A -85,B 0,C 180,E1 -20028.055,E2 -20028.055} C_VEL
LIN {X 0,Y 169.974,Z 205.753,A -85,B 0,C 180,E1 -20027.664,E2 -20027.664} C_VEL
LIN {X 0,Y 167.733,Z 209.43,A -85,B 0,C 180,E1 -20026.673,E2 -20026.673} C_VEL
LIN {X 0,Y 165.587,Z 211.663,A -85,B 0,C 180,E1 -20025.546,E2 -20025.546} C_VEL
LIN {X 0,Y 164.399,Z 215.405,A -85,B 0,C 180,E1 -20025.145,E2 -20025.145} C_VEL
LIN {X 0,Y 160.346,Z 228.889,A -85,B 0,C 180,E1 -20023.762,E2 -20023.762} C_VEL
LIN {X 0,Y 158.548,Z 233.732,A -85,B 0,C 180,E1 -20022.975,E2 -20022.975} C_VEL
LIN {X 0,Y 157.385,Z 235.738,A -85,B 0,C 180,E1 -20022.316,E2 -20022.316} C_VEL
LIN {X 0,Y 156.99,Z 235.462,A -85,B 0,C 180,E1 -20021.969,E2 -20021.969} C_VEL
LIN {X 0,Y 150.293,Z 300.403,A -85,B 0,C 180,E1 -20016.496,E2 -20016.496} C_VEL
LIN {X 0,Y 148.414,Z 316.346,A -85,B 0,C 180,E1 -20014.629,E2 -20014.629} C_VEL
LIN {X 0,Y 146.201,Z 331.602,A -85,B 0,C 180,E1 -20012.331,E2 -20012.331} C_VEL
LIN {X 0,Y 143.638,Z 347.491,A -85,B 0,C 180,E1 -20009.295,E2 -20009.295} C_VEL
LIN {X 0,Y 141.163,Z 362.289,A -85,B 0,C 180,E1 -20005.77,E2 -20005.77} C_VEL
LIN {X 0,Y 138.738,Z 376.531,A -85,B 0,C 180,E1 -20001.548,E2 -20001.548} C_VEL
LIN {X 0,Y 136.937,Z 388.705,A -85,B 0,C 180,E1 -19997.165,E2 -19997.165} C_VEL
LIN {X 0,Y 135.77,Z 399.09,A -85,B 0,C 180,E1 -19992.71,E2 -19992.71} C_VEL
LIN {X 0,Y 135.003,Z 408.406,A -85,B 0,C 180,E1 -19987.945,E2 -19987.945} C_VEL
LIN {X 0,Y 134.638,Z 416.541,A -85,B 0,C 180,E1 -19982.993,E2 -19982.993} C_VEL
LIN {X 0,Y 134.69,Z 422.845,A -85,B 0,C 180,E1 -19978.506,E2 -19978.506} C_VEL
LIN {X 0,Y 135.113,Z 429.165,A -85,B 0,C 180,E1 -19973.036,E2 -19973.036} C_VEL
LIN {X 0,Y 136.739,Z 435.325,A -85,B 0,C 180,E1 -19966.628,E2 -19966.628} C_VEL
LIN {X 0,Y 140.631,Z 440.883,A -85,B 0,C 180,E1 -19959.524,E2 -19959.524} C_VEL
LIN {X 0,Y 145.179,Z 444.284,A -85,B 0,C 180,E1 -19954.172,E2 -19954.172} C_VEL
LIN {X 0,Y 154.559,Z 447.756,A -85,B 0,C 180,E1 -19946.931,E2 -19946.931} C_VEL
LIN {X 0,Y 162.44,Z 449.052,A -85,B 0,C 180,E1 -19942.721,E2 -19942.721} C_VEL
LIN {X 0,Y 171.355,Z 449.586,A -85,B 0,C 180,E1 -19938.988,E2 -19938.988} C_VEL
LIN {X 0,Y 176.123,Z 449.554,A -85,B 0,C 180,E1 -19937.285,E2 -19937.285} C_VEL
LIN {X 0,Y 164.736,Z 451.151,A -85,B 0,C 180,E1 -19933.047,E2 -19933.047} C_VEL
LIN {X 0,Y 156.444,Z 451.789,A -85,B 0,C 180,E1 -19928.971,E2 -19928.971} C_VEL
LIN {X 0,Y 146.298,Z 451.428,A -85,B 0,C 180,E1 -19921.899,E2 -19921.899} C_VEL
LIN {X 0,Y 140.378,Z 450.02,A -85,B 0,C 180,E1 -19915.564,E2 -19915.564} C_VEL
LIN {X 0,Y 137.072,Z 455.452,A -85,B 0,C 180,E1 -19911.033,E2 -19911.033} C_VEL
LIN {X 0,Y 134.649,Z 460.784,A -85,B 0,C 180,E1 -19905.128,E2 -19905.128} C_VEL
LIN {X 0,Y 133.586,Z 464.721,A -85,B 0,C 180,E1 -19899.081,E2 -19899.081} C_VEL
LIN {X 0,Y 133.46,Z 467.319,A -85,B 0,C 180,E1 -19893.019,E2 -19893.019} C_VEL
LIN {X 0,Y 133.53,Z 468.137,A -85,B 0,C 180,E1 -19890,E2 -19890} C_VEL
LIN {X 0,Y 133.435,Z 468.852,A -85,B 0,C 180,E1 -19883.953,E2 -19883.953} C_VEL
LIN {X 0,Y 134.061,Z 468.419,A -85,B 0,C 180,E1 -19877.895,E2 -19877.895} C_VEL
LIN {X 0,Y 135.839,Z 466.863,A -85,B 0,C 180,E1 -19871.915,E2 -19871.915} C_VEL
LIN {X 0,Y 138.961,Z 464.178,A -85,B 0,C 180,E1 -19866.134,E2 -19866.134} C_VEL
LIN {X 0,Y 143.467,Z 460.272,A -85,B 0,C 180,E1 -19860.668,E2 -19860.668} C_VEL
LIN {X 0,Y 149.365,Z 455.069,A -85,B 0,C 180,E1 -19855.623,E2 -19855.623} C_VEL
LIN {X 0,Y 151.901,Z 452.874,A -85,B 0,C 180,E1 -19853.85,E2 -19853.85} C_VEL
LIN {X 0,Y 160.494,Z 452.563,A -85,B 0,C 180,E1 -19848.94,E2 -19848.94} C_VEL
LIN {X 0,Y 169.339,Z 451.637,A -85,B 0,C 180,E1 -19845.126,E2 -19845.126} C_VEL
LIN {X 0,Y 176.087,Z 450.564,A -85,B 0,C 180,E1 -19842.726,E2 -19842.726} C_VEL
LIN {X 0,Y 166.783,Z 450.365,A -85,B 0,C 180,E1 -19839.203,E2 -19839.203} C_VEL
LIN {X 0,Y 158.309,Z 449.439,A -85,B 0,C 180,E1 -19835.248,E2 -19835.248} C_VEL
LIN {X 0,Y 151.16,Z 447.657,A -85,B 0,C 180,E1 -19830.758,E2 -19830.758} C_VEL
LIN {X 0,Y 145.208,Z 445.135,A -85,B 0,C 180,E1 -19825.822,E2 -19825.822} C_VEL
LIN {X 0,Y 139.705,Z 440.741,A -85,B 0,C 180,E1 -19819.085,E2 -19819.085} C_VEL
LIN {X 0,Y 136.527,Z 435.754,A -85,B 0,C 180,E1 -19812.825,E2 -19812.825} C_VEL
LIN {X 0,Y 135.758,Z 436.299,A -85,B 0,C 180,E1 -19810.389,E2 -19810.389} C_VEL
LIN {X 0,Y 136.696,Z 436.809,A -85,B 0,C 180,E1 -19802.946,E2 -19802.946} C_VEL
LIN {X 0,Y 141.23,Z 438.913,A -85,B 0,C 180,E1 -19791.413,E2 -19791.413} C_VEL
LIN {X 0,Y 146.135,Z 440.827,A -85,B 0,C 180,E1 -19784.532,E2 -19784.532} C_VEL
LIN {X 0,Y 146.971,Z 441.547,A -85,B 0,C 180,E1 -19783.027,E2 -19783.027} C_VEL
LIN {X 0,Y 147.423,Z 445.24,A -85,B 0,C 180,E1 -19777.972,E2 -19777.972} C_VEL
LIN {X 0,Y 148.784,Z 445.832,A -85,B 0,C 180,E1 -19776.549,E2 -19776.549} C_VEL
LIN {X 0,Y 149.052,Z 445.872,A -85,B 0,C 180,E1 -19776.372,E2 -19776.372} C_VEL
LIN {X 0,Y 147.832,Z 447.664,A -85,B 0,C 180,E1 -19774.591,E2 -19774.591} C_VEL
LIN {X 0,Y 142.155,Z 452.36,A -85,B 0,C 180,E1 -19770.369,E2 -19770.369} C_VEL
LIN {X 0,Y 136.831,Z 456.452,A -85,B 0,C 180,E1 -19765.266,E2 -19765.266} C_VEL
LIN {X 0,Y 133.149,Z 459.007,A -85,B 0,C 180,E1 -19760.698,E2 -19760.698} C_VEL
LIN {X 0,Y 129.688,Z 461.176,A -85,B 0,C 180,E1 -19754.789,E2 -19754.789} C_VEL
LIN {X 0,Y 127.626,Z 462.147,A -85,B 0,C 180,E1 -19749.56,E2 -19749.56} C_VEL
LIN {X 0,Y 126.224,Z 462.27,A -85,B 0,C 180,E1 -19743.363,E2 -19743.363} C_VEL
LIN {X 0,Y 125.723,Z 461.198,A -85,B 0,C 180,E1 -19736.565,E2 -19736.565} C_VEL
LIN {X 0,Y 126.263,Z 458.692,A -85,B 0,C 180,E1 -19729.51,E2 -19729.51} C_VEL
LIN {X 0,Y 127.45,Z 455.922,A -85,B 0,C 180,E1 -19724.368,E2 -19724.368} C_VEL
LIN {X 0,Y 129.878,Z 450.936,A -85,B 0,C 180,E1 -19717.775,E2 -19717.775} C_VEL
LIN {X 0,Y 133.575,Z 444.293,A -85,B 0,C 180,E1 -19711.412,E2 -19711.412} C_VEL
LIN {X 0,Y 137.676,Z 437.311,A -85,B 0,C 180,E1 -19706.342,E2 -19706.342} C_VEL
LIN {X 0,Y 142.81,Z 428.66,A -85,B 0,C 180,E1 -19701.51,E2 -19701.51} C_VEL
LIN {X 0,Y 147.839,Z 419.85,A -85,B 0,C 180,E1 -19697.648,E2 -19697.648} C_VEL
LIN {X 0,Y 153.57,Z 409.1,A -85,B 0,C 180,E1 -19693.959,E2 -19693.959} C_VEL
LIN {X 0,Y 159.532,Z 396.821,A -85,B 0,C 180,E1 -19690.707,E2 -19690.707} C_VEL
LIN {X 0,Y 164.949,Z 384.218,A -85,B 0,C 180,E1 -19688.111,E2 -19688.111} C_VEL
LIN {X 0,Y 169.573,Z 371.822,A -85,B 0,C 180,E1 -19686.099,E2 -19686.099} C_VEL
LIN {X 0,Y 174.225,Z 357.189,A -85,B 0,C 180,E1 -19684.301,E2 -19684.301} C_VEL
LIN {X 0,Y 177.763,Z 342.968,A -85,B 0,C 180,E1 -19682.957,E2 -19682.957} C_VEL
LIN {X 0,Y 180.599,Z 327.902,A -85,B 0,C 180,E1 -19681.925,E2 -19681.925} C_VEL
LIN {X 0,Y 182.8,Z 311.041,A -85,B 0,C 180,E1 -19681.198,E2 -19681.198} C_VEL
LIN {X 0,Y 188.796,Z 241.455,A -85,B 0,C 180,E1 -19678.96,E2 -19678.96} C_VEL
LIN {X 0,Y 184.638,Z 231.846,A -85,B 0,C 180,E1 -19676.749,E2 -19676.749} C_VEL
LIN {X 0,Y 179.737,Z 221.737,A -85,B 0,C 180,E1 -19673.957,E2 -19673.957} C_VEL
LIN {X 0,Y 174.543,Z 212.044,A -85,B 0,C 180,E1 -19670.723,E2 -19670.723} C_VEL
LIN {X 0,Y 173.235,Z 209.871,A -85,B 0,C 180,E1 -19669.859,E2 -19669.859} C_VEL
LIN {X 0,Y 172.233,Z 210.377,A -85,B 0,C 180,E1 -19669.36,E2 -19669.36} C_VEL
LIN {X 0,Y 169.205,Z 215.052,A -85,B 0,C 180,E1 -19668.059,E2 -19668.059} C_VEL
LIN {X 0,Y 167.666,Z 216.745,A -85,B 0,C 180,E1 -19667.31,E2 -19667.31} C_VEL
LIN {X 0,Y 162.981,Z 231.817,A -85,B 0,C 180,E1 -19665.855,E2 -19665.855} C_VEL
LIN {X 0,Y 160.778,Z 237.568,A -85,B 0,C 180,E1 -19664.979,E2 -19664.979} C_VEL
LIN {X 0,Y 158.84,Z 241.182,A -85,B 0,C 180,E1 -19664.01,E2 -19664.01} C_VEL
LIN {X 0,Y 153.547,Z 262.625,A -85,B 0,C 180,E1 -19662.465,E2 -19662.465} C_VEL
LIN {X 0,Y 148.732,Z 280.011,A -85,B 0,C 180,E1 -19660.67,E2 -19660.67} C_VEL
LIN {X 0,Y 146,Z 288.321,A -85,B 0,C 180,E1 -19659.331,E2 -19659.331} C_VEL
LIN {X 0,Y 145.155,Z 290.138,A -85,B 0,C 180,E1 -19658.786,E2 -19658.786} C_VEL
LIN {X 0,Y 144.764,Z 290.539,A -85,B 0,C 180,E1 -19658.465,E2 -19658.465} C_VEL
LIN {X 0,Y 144.531,Z 290.329,A -85,B 0,C 180,E1 -19658.205,E2 -19658.205} C_VEL
LIN {X 0,Y 144.424,Z 289.764,A -85,B 0,C 180,E1 -19658.017,E2 -19658.017} C_VEL
LIN {X 0,Y 142.27,Z 309.618,A -85,B 0,C 180,E1 -19655.918,E2 -19655.918} C_VEL
LIN {X 0,Y 139.943,Z 326.235,A -85,B 0,C 180,E1 -19653.535,E2 -19653.535} C_VEL
LIN {X 0,Y 137.255,Z 343.277,A -85,B 0,C 180,E1 -19650.332,E2 -19650.332} C_VEL
LIN {X 0,Y 134.468,Z 359.301,A -85,B 0,C 180,E1 -19646.51,E2 -19646.51} C_VEL
LIN {X 0,Y 132.07,Z 373.463,A -85,B 0,C 180,E1 -19642.282,E2 -19642.282} C_VEL
LIN {X 0,Y 130.02,Z 387.097,A -85,B 0,C 180,E1 -19637.296,E2 -19637.296} C_VEL
LIN {X 0,Y 128.838,Z 397.657,A -85,B 0,C 180,E1 -19632.604,E2 -19632.604} C_VEL
LIN {X 0,Y 128.001,Z 408.101,A -85,B 0,C 180,E1 -19627.044,E2 -19627.044} C_VEL
LIN {X 0,Y 127.725,Z 415.554,A -85,B 0,C 180,E1 -19622.366,E2 -19622.366} C_VEL
LIN {X 0,Y 127.885,Z 422.837,A -85,B 0,C 180,E1 -19616.851,E2 -19616.851} C_VEL
LIN {X 0,Y 128.301,Z 428.161,A -85,B 0,C 180,E1 -19612.13,E2 -19612.13} C_VEL
LIN {X 0,Y 130.62,Z 435.377,A -85,B 0,C 180,E1 -19604.395,E2 -19604.395} C_VEL
LIN {X 0,Y 134.072,Z 439.98,A -85,B 0,C 180,E1 -19598.474,E2 -19598.474} C_VEL
LIN {X 0,Y 138.841,Z 443.662,A -85,B 0,C 180,E1 -19592.899,E2 -19592.899} C_VEL
LIN {X 0,Y 145.062,Z 446.518,A -85,B 0,C 180,E1 -19587.797,E2 -19587.797} C_VEL
LIN {X 0,Y 152.622,Z 448.555,A -85,B 0,C 180,E1 -19583.229,E2 -19583.229} C_VEL
LIN {X 0,Y 161.334,Z 449.823,A -85,B 0,C 180,E1 -19579.2,E2 -19579.2} C_VEL
LIN {X 0,Y 166.083,Z 450.155,A -85,B 0,C 180,E1 -19577.387,E2 -19577.387} C_VEL
LIN {X 0,Y 155.136,Z 450.989,A -85,B 0,C 180,E1 -19572.807,E2 -19572.807} C_VEL
LIN {X 0,Y 143.587,Z 450.688,A -85,B 0,C 180,E1 -19565.969,E2 -19565.969} C_VEL
LIN {X 0,Y 134.965,Z 448.812,A -85,B 0,C 180,E1 -19557.947,E2 -19557.947} C_VEL
LIN {X 0,Y 134.549,Z 448.662,A -85,B 0,C 180,E1 -19557.409,E2 -19557.409} C_VEL
LIN {X 0,Y 130.435,Z 454.863,A -85,B 0,C 180,E1 -19552.159,E2 -19552.159} C_VEL
LIN {X 0,Y 127.746,Z 460.287,A -85,B 0,C 180,E1 -19545.967,E2 -19545.967} C_VEL
LIN {X 0,Y 126.541,Z 464.302,A -85,B 0,C 180,E1 -19539.591,E2 -19539.591} C_VEL
LIN {X 0,Y 126.369,Z 466.985,A -85,B 0,C 180,E1 -19533.188,E2 -19533.188} C_VEL
LIN {X 0,Y 126.443,Z 467.846,A -85,B 0,C 180,E1 -19530,E2 -19530} C_VEL
LIN {X 0,Y 126.351,Z 468.644,A -85,B 0,C 180,E1 -19523.613,E2 -19523.613} C_VEL
LIN {X 0,Y 127.061,Z 468.296,A -85,B 0,C 180,E1 -19517.218,E2 -19517.218} C_VEL
LIN {X 0,Y 129.05,Z 466.836,A -85,B 0,C 180,E1 -19510.928,E2 -19510.928} C_VEL
LIN {X 0,Y 132.428,Z 464.216,A -85,B 0,C 180,E1 -19504.877,E2 -19504.877} C_VEL
LIN {X 0,Y 137.285,Z 460.39,A -85,B 0,C 180,E1 -19499.208,E2 -19499.208} C_VEL
LIN {X 0,Y 143.549,Z 455.305,A -85,B 0,C 180,E1 -19494.02,E2 -19494.02} C_VEL
LIN {X 0,Y 147.653,Z 451.985,A -85,B 0,C 180,E1 -19491.338,E2 -19491.338} C_VEL
LIN {X 0,Y 155.213,Z 452.004,A -85,B 0,C 180,E1 -19487.219,E2 -19487.219} C_VEL
LIN {X 0,Y 164.383,Z 451.366,A -85,B 0,C 180,E1 -19483.38,E2 -19483.38} C_VEL
LIN {X 0,Y 166.016,Z 451.15,A -85,B 0,C 180,E1 -19482.635,E2 -19482.635} C_VEL
LIN {X 0,Y 156.803,Z 450.26,A -85,B 0,C 180,E1 -19478.864,E2 -19478.864} C_VEL
LIN {X 0,Y 148.69,Z 448.526,A -85,B 0,C 180,E1 -19474.554,E2 -19474.554} C_VEL
LIN {X 0,Y 141.824,Z 446.087,A -85,B 0,C 180,E1 -19469.705,E2 -19469.705} C_VEL
LIN {X 0,Y 134.112,Z 440.834,A -85,B 0,C 180,E1 -19461.519,E2 -19461.519} C_VEL
LIN {X 0,Y 132.608,Z 439.249,A -85,B 0,C 180,E1 -19459.343,E2 -19459.343} C_VEL
LIN {X 0,Y 130.818,Z 439.731,A -85,B 0,C 180,E1 -19455.581,E2 -19455.581} C_VEL
LIN {X 0,Y 130.304,Z 439.798,A -85,B 0,C 180,E1 -19452.458,E2 -19452.458} C_VEL
LIN {X 0,Y 129.958,Z 440.369,A -85,B 0,C 180,E1 -19446.208,E2 -19446.208} C_VEL
LIN {X 0,Y 130.601,Z 440.559,A -85,B 0,C 180,E1 -19443.084,E2 -19443.084} C_VEL
LIN {X 0,Y 135.383,Z 442.548,A -85,B 0,C 180,E1 -19430.514,E2 -19430.514} C_VEL
LIN {X 0,Y 144.086,Z 445.043,A -85,B 0,C 180,E1 -19420.035,E2 -19420.035} C_VEL
LIN {X 0,Y 148.784,Z 445.832,A -85,B 0,C 180,E1 -19416.549,E2 -19416.549} C_VEL
LIN {X 0,Y 149.021,Z 446.291,A -85,B 0,C 180,E1 -19415.862,E2 -19415.862} C_VEL
LIN {X 0,Y 148.024,Z 447.278,A -85,B 0,C 180,E1 -19415.039,E2 -19415.039} C_VEL
LIN {X 0,Y 145.386,Z 448.895,A -85,B 0,C 180,E1 -19414.098,E2 -19414.098} C_VEL
LIN {X 0,Y 137.248,Z 452.627,A -85,B 0,C 180,E1 -19412.101,E2 -19412.101} C_VEL
LIN {X 0,Y 134.917,Z 453.908,A -85,B 0,C 180,E1 -19410.887,E2 -19410.887} C_VEL
LIN {X 0,Y 128.922,Z 458.014,A -85,B 0,C 180,E1 -19404.856,E2 -19404.856} C_VEL
LIN {X 0,Y 126.151,Z 459.732,A -85,B 0,C 180,E1 -19401.257,E2 -19401.257} C_VEL
LIN {X 0,Y 123.484,Z 461.224,A -85,B 0,C 180,E1 -19396.922,E2 -19396.922} C_VEL
LIN {X 0,Y 120.57,Z 462.449,A -85,B 0,C 180,E1 -19389.88,E2 -19389.88} C_VEL
LIN {X 0,Y 119.258,Z 462.473,A -85,B 0,C 180,E1 -19384.406,E2 -19384.406} C_VEL
LIN {X 0,Y 118.621,Z 461.45,A -85,B 0,C 180,E1 -19377.285,E2 -19377.285} C_VEL
LIN {X 0,Y 118.959,Z 459.409,A -85,B 0,C 180,E1 -19370.761,E2 -19370.761} C_VEL
LIN {X 0,Y 120.039,Z 456.77,A -85,B 0,C 180,E1 -19365.276,E2 -19365.276} C_VEL
LIN {X 0,Y 122.459,Z 452.032,A -85,B 0,C 180,E1 -19358.249,E2 -19358.249} C_VEL
LIN {X 0,Y 125.838,Z 446.098,A -85,B 0,C 180,E1 -19351.874,E2 -19351.874} C_VEL
LIN {X 0,Y 130.274,Z 438.945,A -85,B 0,C 180,E1 -19346.133,E2 -19346.133} C_VEL
LIN {X 0,Y 135.434,Z 430.619,A -85,B 0,C 180,E1 -19341.044,E2 -19341.044} C_VEL
LIN {X 0,Y 140.611,Z 422.066,A -85,B 0,C 180,E1 -19337.002,E2 -19337.002} C_VEL
LIN {X 0,Y 146.348,Z 411.981,A -85,B 0,C 180,E1 -19333.254,E2 -19333.254} C_VEL
LIN {X 0,Y 152.05,Z 401.03,A -85,B 0,C 180,E1 -19330.069,E2 -19330.069} C_VEL
LIN {X 0,Y 157.55,Z 389.228,A -85,B 0,C 180,E1 -19327.372,E2 -19327.372} C_VEL
LIN {X 0,Y 162.62,Z 376.913,A -85,B 0,C 180,E1 -19325.173,E2 -19325.173} C_VEL
LIN {X 0,Y 167.613,Z 362.632,A -85,B 0,C 180,E1 -19323.208,E2 -19323.208} C_VEL
LIN {X 0,Y 171.651,Z 348.491,A -85,B 0,C 180,E1 -19321.744,E2 -19321.744} C_VEL
LIN {X 0,Y 174.789,Z 333.778,A -85,B 0,C 180,E1 -19320.574,E2 -19320.574} C_VEL
LIN {X 0,Y 177.19,Z 318.714,A -85,B 0,C 180,E1 -19319.786,E2 -19319.786} C_VEL
LIN {X 0,Y 180.857,Z 280.465,A -85,B 0,C 180,E1 -19318.522,E2 -19318.522} C_VEL
LIN {X 0,Y 184.106,Z 244.036,A -85,B 0,C 180,E1 -19317.357,E2 -19317.357} C_VEL
LIN {X 0,Y 179.494,Z 233.381,A -85,B 0,C 180,E1 -19314.703,E2 -19314.703} C_VEL
LIN {X 0,Y 174.909,Z 223.894,A -85,B 0,C 180,E1 -19311.857,E2 -19311.857} C_VEL
LIN {X 0,Y 172.411,Z 218.972,A -85,B 0,C 180,E1 -19310.184,E2 -19310.184} C_VEL
LIN {X 0,Y 171.94,Z 219.074,A -85,B 0,C 180,E1 -19309.942,E2 -19309.942} C_VEL
LIN {X 0,Y 170.015,Z 221.58,A -85,B 0,C 180,E1 -19309.105,E2 -19309.105} C_VEL
LIN {X 0,Y 165.84,Z 234.736,A -85,B 0,C 180,E1 -19307.884,E2 -19307.884} C_VEL
LIN {X 0,Y 163.223,Z 241.345,A -85,B 0,C 180,E1 -19306.931,E2 -19306.931} C_VEL
LIN {X 0,Y 161.265,Z 245.281,A -85,B 0,C 180,E1 -19306.079,E2 -19306.079} C_VEL
LIN {X 0,Y 155.58,Z 267.51,A -85,B 0,C 180,E1 -19304.526,E2 -19304.526} C_VEL
LIN {X 0,Y 151.108,Z 283.011,A -85,B 0,C 180,E1 -19302.946,E2 -19302.946} C_VEL
LIN {X 0,Y 148.058,Z 291.861,A -85,B 0,C 180,E1 -19301.584,E2 -19301.584} C_VEL
LIN {X 0,Y 146.099,Z 295.819,A -85,B 0,C 180,E1 -19300.42,E2 -19300.42} C_VEL
LIN {X 0,Y 145.72,Z 296.498,A -85,B 0,C 180,E1 -19300.173,E2 -19300.173} C_VEL
LIN {X 0,Y 142.245,Z 310.245,A -85,B 0,C 180,E1 -19298.82,E2 -19298.82} C_VEL
LIN {X 0,Y 138.719,Z 321.546,A -85,B 0,C 180,E1 -19297.215,E2 -19297.215} C_VEL
LIN {X 0,Y 135.926,Z 328.352,A -85,B 0,C 180,E1 -19295.798,E2 -19295.798} C_VEL
LIN {X 0,Y 133.393,Z 333.428,A -85,B 0,C 180,E1 -19294.271,E2 -19294.271} C_VEL
LIN {X 0,Y 132.129,Z 335.215,A -85,B 0,C 180,E1 -19293.267,E2 -19293.267} C_VEL
LIN {X 0,Y 131.391,Z 335.233,A -85,B 0,C 180,E1 -19292.151,E2 -19292.151} C_VEL
LIN {X 0,Y 129.015,Z 349.337,A -85,B 0,C 180,E1 -19289.047,E2 -19289.047} C_VEL
LIN {X 0,Y 126.521,Z 364.013,A -85,B 0,C 180,E1 -19285.06,E2 -19285.06} C_VEL
LIN {X 0,Y 124.32,Z 377.02,A -85,B 0,C 180,E1 -19280.692,E2 -19280.692} C_VEL
LIN {X 0,Y 122.666,Z 389.084,A -85,B 0,C 180,E1 -19275.793,E2 -19275.793} C_VEL
LIN {X 0,Y 121.607,Z 399.51,A -85,B 0,C 180,E1 -19270.742,E2 -19270.742} C_VEL
LIN {X 0,Y 121.003,Z 408.053,A -85,B 0,C 180,E1 -19265.835,E2 -19265.835} C_VEL
LIN {X 0,Y 120.867,Z 415.49,A -85,B 0,C 180,E1 -19260.834,E2 -19260.834} C_VEL
LIN {X 0,Y 121.17,Z 422.794,A -85,B 0,C 180,E1 -19255.01,E2 -19255.01} C_VEL
LIN {X 0,Y 122.679,Z 431.159,A -85,B 0,C 180,E1 -19246.754,E2 -19246.754} C_VEL
LIN {X 0,Y 126.505,Z 437.769,A -85,B 0,C 180,E1 -19238.833,E2 -19238.833} C_VEL
LIN {X 0,Y 132.603,Z 442.888,A -85,B 0,C 180,E1 -19231.511,E2 -19231.511} C_VEL
LIN {X 0,Y 139.115,Z 446.065,A -85,B 0,C 180,E1 -19226.241,E2 -19226.241} C_VEL
LIN {X 0,Y 147.019,Z 448.426,A -85,B 0,C 180,E1 -19221.579,E2 -19221.579} C_VEL
LIN {X 0,Y 156.034,Z 450.079,A -85,B 0,C 180,E1 -19217.498,E2 -19217.498} C_VEL
LIN {X 0,Y 154.692,Z 450.183,A -85,B 0,C 180,E1 -19216.628,E2 -19216.628} C_VEL
LIN {X 0,Y 145.72,Z 450.127,A -85,B 0,C 180,E1 -19212.471,E2 -19212.471} C_VEL
LIN {X 0,Y 137.952,Z 449.472,A -85,B 0,C 180,E1 -19207.687,E2 -19207.687} C_VEL
LIN {X 0,Y 129.021,Z 447.259,A -85,B 0,C 180,E1 -19199.581,E2 -19199.581} C_VEL
LIN {X 0,Y 128.847,Z 447.221,A -85,B 0,C 180,E1 -19199.4,E2 -19199.4} C_VEL
LIN {X 0,Y 124.887,Z 452.632,A -85,B 0,C 180,E1 -19194.965,E2 -19194.965} C_VEL
LIN {X 0,Y 121.493,Z 458.519,A -85,B 0,C 180,E1 -19188.552,E2 -19188.552} C_VEL
LIN {X 0,Y 120.022,Z 461.994,A -85,B 0,C 180,E1 -19183.546,E2 -19183.546} C_VEL
LIN {X 0,Y 119.255,Z 465.423,A -85,B 0,C 180,E1 -19176.769,E2 -19176.769} C_VEL
LIN {X 0,Y 119.273,Z 466.647,A -85,B 0,C 180,E1 -19173.378,E2 -19173.378} C_VEL
LIN {X 0,Y 119.358,Z 467.552,A -85,B 0,C 180,E1 -19170,E2 -19170} C_VEL
LIN {X 0,Y 119.26,Z 468.433,A -85,B 0,C 180,E1 -19163.231,E2 -19163.231} C_VEL
LIN {X 0,Y 120.092,Z 468.177,A -85,B 0,C 180,E1 -19156.462,E2 -19156.462} C_VEL
LIN {X 0,Y 122.308,Z 466.793,A -85,B 0,C 180,E1 -19149.832,E2 -19149.832} C_VEL
LIN {X 0,Y 126.602,Z 463.824,A -85,B 0,C 180,E1 -19142.646,E2 -19142.646} C_VEL
LIN {X 0,Y 132.753,Z 459.443,A -85,B 0,C 180,E1 -19136.229,E2 -19136.229} C_VEL
LIN {X 0,Y 139.696,Z 454.151,A -85,B 0,C 180,E1 -19131.033,E2 -19131.033} C_VEL
LIN {X 0,Y 143.726,Z 451.043,A -85,B 0,C 180,E1 -19128.69,E2 -19128.69} C_VEL
LIN {X 0,Y 154.763,Z 451.172,A -85,B 0,C 180,E1 -19123.399,E2 -19123.399} C_VEL
LIN {X 0,Y 156.064,Z 451.052,A -85,B 0,C 180,E1 -19122.491,E2 -19122.491} C_VEL
LIN {X 0,Y 146.944,Z 449.358,A -85,B 0,C 180,E1 -19118.444,E2 -19118.444} C_VEL
LIN {X 0,Y 139.154,Z 446.971,A -85,B 0,C 180,E1 -19113.748,E2 -19113.748} C_VEL
LIN {X 0,Y 130.931,Z 442.662,A -85,B 0,C 180,E1 -19106.714,E2 -19106.714} C_VEL
LIN {X 0,Y 127.775,Z 443.035,A -85,B 0,C 180,E1 -19102.644,E2 -19102.644} C_VEL
LIN {X 0,Y 125.558,Z 443.205,A -85,B 0,C 180,E1 -19097.906,E2 -19097.906} C_VEL
LIN {X 0,Y 124.376,Z 444.044,A -85,B 0,C 180,E1 -19083.238,E2 -19083.238} C_VEL
LIN {X 0,Y 128.888,Z 445.688,A -85,B 0,C 180,E1 -19070.584,E2 -19070.584} C_VEL
LIN {X 0,Y 138.049,Z 448.04,A -85,B 0,C 180,E1 -19059.122,E2 -19059.122} C_VEL
LIN {X 0,Y 141.33,Z 448.525,A -85,B 0,C 180,E1 -19056.557,E2 -19056.557} C_VEL
LIN {X 0,Y 139.901,Z 450.216,A -85,B 0,C 180,E1 -19054.721,E2 -19054.721} C_VEL
LIN {X 0,Y 134.917,Z 453.908,A -85,B 0,C 180,E1 -19050.887,E2 -19050.887} C_VEL
LIN {X 0,Y 131.913,Z 455.69,A -85,B 0,C 180,E1 -19048.837,E2 -19048.837} C_VEL
LIN {X 0,Y 125.727,Z 458.27,A -85,B 0,C 180,E1 -19045.581,E2 -19045.581} C_VEL
LIN {X 0,Y 120.92,Z 459.949,A -85,B 0,C 180,E1 -19042.739,E2 -19042.739} C_VEL
LIN {X 0,Y 118.167,Z 460.92,A -85,B 0,C 180,E1 -19040.273,E2 -19040.273} C_VEL
LIN {X 0,Y 117.53,Z 461.203,A -85,B 0,C 180,E1 -19039.376,E2 -19039.376} C_VEL
LIN {X 0,Y 114.223,Z 462.508,A -85,B 0,C 180,E1 -19032.407,E2 -19032.407} C_VEL
LIN {X 0,Y 112.122,Z 462.609,A -85,B 0,C 180,E1 -19024.342,E2 -19024.342} C_VEL
LIN {X 0,Y 111.53,Z 461.701,A -85,B 0,C 180,E1 -19018.088,E2 -19018.088} C_VEL
LIN {X 0,Y 111.995,Z 459.126,A -85,B 0,C 180,E1 -19009.727,E2 -19009.727} C_VEL
LIN {X 0,Y 113.702,Z 455.505,A -85,B 0,C 180,E1 -19002.494,E2 -19002.494} C_VEL
LIN {X 0,Y 116.588,Z 450.274,A -85,B 0,C 180,E1 -18995.188,E2 -18995.188} C_VEL
LIN {X 0,Y 120.916,Z 443.474,A -85,B 0,C 180,E1 -18988.335,E2 -18988.335} C_VEL
LIN {X 0,Y 125.751,Z 436.076,A -85,B 0,C 180,E1 -18982.776,E2 -18982.776} C_VEL
LIN {X 0,Y 131.626,Z 427.087,A -85,B 0,C 180,E1 -18977.668,E2 -18977.668} C_VEL
LIN {X 0,Y 137.269,Z 417.901,A -85,B 0,C 180,E1 -18973.645,E2 -18973.645} C_VEL
LIN {X 0,Y 143.515,Z 406.99,A -85,B 0,C 180,E1 -18969.953,E2 -18969.953} C_VEL
LIN {X 0,Y 149.642,Z 395.061,A -85,B 0,C 180,E1 -18966.838,E2 -18966.838} C_VEL
LIN {X 0,Y 155.184,Z 382.863,A -85,B 0,C 180,E1 -18964.373,E2 -18964.373} C_VEL
LIN {X 0,Y 160.439,Z 369.379,A -85,B 0,C 180,E1 -18962.262,E2 -18962.262} C_VEL
LIN {X 0,Y 165.205,Z 354.697,A -85,B 0,C 180,E1 -18960.536,E2 -18960.536} C_VEL
LIN {X 0,Y 168.997,Z 339.596,A -85,B 0,C 180,E1 -18959.2,E2 -18959.2} C_VEL
LIN {X 0,Y 171.739,Z 324.922,A -85,B 0,C 180,E1 -18958.291,E2 -18958.291} C_VEL
LIN {X 0,Y 173.794,Z 308.714,A -85,B 0,C 180,E1 -18957.664,E2 -18957.664} C_VEL
LIN {X 0,Y 179.53,Z 246.595,A -85,B 0,C 180,E1 -18955.67,E2 -18955.67} C_VEL
LIN {X 0,Y 173.813,Z 233.431,A -85,B 0,C 180,E1 -18952.074,E2 -18952.074} C_VEL
LIN {X 0,Y 171.654,Z 229.113,A -85,B 0,C 180,E1 -18950.633,E2 -18950.633} C_VEL
LIN {X 0,Y 168.441,Z 238.706,A -85,B 0,C 180,E1 -18949.727,E2 -18949.727} C_VEL
LIN {X 0,Y 165.643,Z 245.481,A -85,B 0,C 180,E1 -18948.746,E2 -18948.746} C_VEL
LIN {X 0,Y 164.025,Z 248.873,A -85,B 0,C 180,E1 -18948.115,E2 -18948.115} C_VEL
LIN {X 0,Y 158.586,Z 269.49,A -85,B 0,C 180,E1 -18946.758,E2 -18946.758} C_VEL
LIN {X 0,Y 153.64,Z 286.095,A -85,B 0,C 180,E1 -18945.156,E2 -18945.156} C_VEL
LIN {X 0,Y 150.396,Z 295.29,A -85,B 0,C 180,E1 -18943.805,E2 -18943.805} C_VEL
LIN {X 0,Y 147.772,Z 300.8,A -85,B 0,C 180,E1 -18942.436,E2 -18942.436} C_VEL
LIN {X 0,Y 143.873,Z 315.137,A -85,B 0,C 180,E1 -18941.027,E2 -18941.027} C_VEL
LIN {X 0,Y 139.947,Z 326.199,A -85,B 0,C 180,E1 -18939.465,E2 -18939.465} C_VEL
LIN {X 0,Y 136.684,Z 333.268,A -85,B 0,C 180,E1 -18937.983,E2 -18937.983} C_VEL
LIN {X 0,Y 133.782,Z 338.388,A -85,B 0,C 180,E1 -18936.463,E2 -18936.463} C_VEL
LIN {X 0,Y 132.585,Z 340.067,A -85,B 0,C 180,E1 -18935.669,E2 -18935.669} C_VEL
LIN {X 0,Y 130.923,Z 341.781,A -85,B 0,C 180,E1 -18934.309,E2 -18934.309} C_VEL
LIN {X 0,Y 126.131,Z 350.699,A -85,B 0,C 180,E1 -18931.962,E2 -18931.962} C_VEL
LIN {X 0,Y 123.327,Z 355.105,A -85,B 0,C 180,E1 -18930.195,E2 -18930.195} C_VEL
LIN {X 0,Y 121.87,Z 356.997,A -85,B 0,C 180,E1 -18929.023,E2 -18929.023} C_VEL
LIN {X 0,Y 120.731,Z 358.195,A -85,B 0,C 180,E1 -18927.757,E2 -18927.757} C_VEL
LIN {X 0,Y 120.322,Z 358.029,A -85,B 0,C 180,E1 -18926.683,E2 -18926.683} C_VEL
LIN {X 0,Y 117.833,Z 372.568,A -85,B 0,C 180,E1 -18921.888,E2 -18921.888} C_VEL
LIN {X 0,Y 115.977,Z 385.334,A -85,B 0,C 180,E1 -18916.73,E2 -18916.73} C_VEL
LIN {X 0,Y 114.828,Z 396.302,A -85,B 0,C 180,E1 -18911.384,E2 -18911.384} C_VEL
LIN {X 0,Y 114.134,Z 406.631,A -85,B 0,C 180,E1 -18905.301,E2 -18905.301} C_VEL
LIN {X 0,Y 114.059,Z 414.226,A -85,B 0,C 180,E1 -18900.001,E2 -18900.001} C_VEL
LIN {X 0,Y 114.368,Z 420.688,A -85,B 0,C 180,E1 -18894.712,E2 -18894.712} C_VEL
LIN {X 0,Y 115.438,Z 427.852,A -85,B 0,C 180,E1 -18887.698,E2 -18887.698} C_VEL
LIN {X 0,Y 118.123,Z 433.835,A -85,B 0,C 180,E1 -18880.9,E2 -18880.9} C_VEL
LIN {X 0,Y 123.608,Z 439.906,A -85,B 0,C 180,E1 -18872.945,E2 -18872.945} C_VEL
LIN {X 0,Y 129.716,Z 443.781,A -85,B 0,C 180,E1 -18867.195,E2 -18867.195} C_VEL
LIN {X 0,Y 137.243,Z 446.875,A -85,B 0,C 180,E1 -18862.086,E2 -18862.086} C_VEL
LIN {X 0,Y 146.095,Z 449.202,A -85,B 0,C 180,E1 -18857.665,E2 -18857.665} C_VEL
LIN {X 0,Y 145.099,Z 449.29,A -85,B 0,C 180,E1 -18856.597,E2 -18856.597} C_VEL
LIN {X 0,Y 136.336,Z 448.656,A -85,B 0,C 180,E1 -18852.078,E2 -18852.078} C_VEL
LIN {X 0,Y 128.909,Z 447.419,A -85,B 0,C 180,E1 -18846.849,E2 -18846.849} C_VEL
LIN {X 0,Y 123.375,Z 445.723,A -85,B 0,C 180,E1 -18841.558,E2 -18841.558} C_VEL
LIN {X 0,Y 118.46,Z 451.981,A -85,B 0,C 180,E1 -18836.421,E2 -18836.421} C_VEL
LIN {X 0,Y 114.74,Z 457.972,A -85,B 0,C 180,E1 -18829.687,E2 -18829.687} C_VEL
LIN {X 0,Y 113.088,Z 461.497,A -85,B 0,C 180,E1 -18824.394,E2 -18824.394} C_VEL
LIN {X 0,Y 112.187,Z 465.025,A -85,B 0,C 180,E1 -18817.198,E2 -18817.198} C_VEL
LIN {X 0,Y 112.161,Z 466.297,A -85,B 0,C 180,E1 -18813.593,E2 -18813.593} C_VEL
LIN {X 0,Y 112.259,Z 467.25,A -85,B 0,C 180,E1 -18810,E2 -18810} C_VEL
LIN {X 0,Y 112.196,Z 468.223,A -85,B 0,C 180,E1 -18802.803,E2 -18802.803} C_VEL
LIN {X 0,Y 113.155,Z 468.056,A -85,B 0,C 180,E1 -18795.615,E2 -18795.615} C_VEL
LIN {X 0,Y 115.621,Z 466.727,A -85,B 0,C 180,E1 -18788.61,E2 -18788.61} C_VEL
LIN {X 0,Y 119.962,Z 464.067,A -85,B 0,C 180,E1 -18781.494,E2 -18781.494} C_VEL
LIN {X 0,Y 126.905,Z 459.617,A -85,B 0,C 180,E1 -18774.445,E2 -18774.445} C_VEL
LIN {X 0,Y 134.245,Z 454.421,A -85,B 0,C 180,E1 -18769.126,E2 -18769.126} C_VEL
LIN {X 0,Y 140.39,Z 450.051,A -85,B 0,C 180,E1 -18765.756,E2 -18765.756} C_VEL
LIN {X 0,Y 145.177,Z 450.278,A -85,B 0,C 180,E1 -18763.436,E2 -18763.436} C_VEL
LIN {X 0,Y 146.034,Z 450.156,A -85,B 0,C 180,E1 -18762.357,E2 -18762.357} C_VEL
LIN {X 0,Y 137.255,Z 447.804,A -85,B 0,C 180,E1 -18757.911,E2 -18757.911} C_VEL
LIN {X 0,Y 131.953,Z 445.915,A -85,B 0,C 180,E1 -18754.464,E2 -18754.464} C_VEL
LIN {X 0,Y 126.782,Z 446.262,A -85,B 0,C 180,E1 -18749.926,E2 -18749.926} C_VEL
LIN {X 0,Y 117.481,Z 447.167,A -85,B 0,C 180,E1 -18726.871,E2 -18726.871} C_VEL
LIN {X 0,Y 118.015,Z 447.285,A -85,B 0,C 180,E1 -18723.413,E2 -18723.413} C_VEL
LIN {X 0,Y 122.538,Z 448.727,A -85,B 0,C 180,E1 -18710.091,E2 -18710.091} C_VEL
LIN {X 0,Y 133.541,Z 450.992,A -85,B 0,C 180,E1 -18696.801,E2 -18696.801} C_VEL
LIN {X 0,Y 131.764,Z 452.69,A -85,B 0,C 180,E1 -18694.74,E2 -18694.74} C_VEL
LIN {X 0,Y 125.954,Z 456.485,A -85,B 0,C 180,E1 -18689.854,E2 -18689.854} C_VEL
LIN {X 0,Y 120.994,Z 459.406,A -85,B 0,C 180,E1 -18684.41,E2 -18684.41} C_VEL
LIN {X 0,Y 117.53,Z 461.203,A -85,B 0,C 180,E1 -18679.376,E2 -18679.376} C_VEL
LIN {X 0,Y 115.368,Z 461.945,A -85,B 0,C 180,E1 -18676.698,E2 -18676.698} C_VEL
LIN {X 0,Y 110.557,Z 462.708,A -85,B 0,C 180,E1 -18672.317,E2 -18672.317} C_VEL
LIN {X 0,Y 106.953,Z 462.931,A -85,B 0,C 180,E1 -18668.566,E2 -18668.566} C_VEL
LIN {X 0,Y 105.237,Z 462.804,A -85,B 0,C 180,E1 -18665.491,E2 -18665.491} C_VEL
LIN {X 0,Y 104.972,Z 462.664,A -85,B 0,C 180,E1 -18664.422,E2 -18664.422} C_VEL
LIN {X 0,Y 104.44,Z 461.753,A -85,B 0,C 180,E1 -18658.102,E2 -18658.102} C_VEL
LIN {X 0,Y 104.921,Z 459.224,A -85,B 0,C 180,E1 -18649.568,E2 -18649.568} C_VEL
LIN {X 0,Y 106.862,Z 455.292,A -85,B 0,C 180,E1 -18641.379,E2 -18641.379} C_VEL
LIN {X 0,Y 109.142,Z 451.429,A -85,B 0,C 180,E1 -18635.543,E2 -18635.543} C_VEL
LIN {X 0,Y 112.453,Z 446.326,A -85,B 0,C 180,E1 -18629.628,E2 -18629.628} C_VEL
LIN {X 0,Y 117.61,Z 438.885,A -85,B 0,C 180,E1 -18623.136,E2 -18623.136} C_VEL
LIN {X 0,Y 123.671,Z 430.138,A -85,B 0,C 180,E1 -18617.499,E2 -18617.499} C_VEL
LIN {X 0,Y 130.214,Z 420.223,A -85,B 0,C 180,E1 -18612.732,E2 -18612.732} C_VEL
LIN {X 0,Y 136.629,Z 409.717,A -85,B 0,C 180,E1 -18608.895,E2 -18608.895} C_VEL
LIN {X 0,Y 142.904,Z 398.28,A -85,B 0,C 180,E1 -18605.677,E2 -18605.677} C_VEL
LIN {X 0,Y 148.977,Z 385.83,A -85,B 0,C 180,E1 -18602.996,E2 -18602.996} C_VEL
LIN {X 0,Y 154.632,Z 372.244,A -85,B 0,C 180,E1 -18600.745,E2 -18600.745} C_VEL
LIN {X 0,Y 159.547,Z 358.252,A -85,B 0,C 180,E1 -18599.014,E2 -18599.014} C_VEL
LIN {X 0,Y 163.478,Z 344.135,A -85,B 0,C 180,E1 -18597.677,E2 -18597.677} C_VEL
LIN {X 0,Y 166.573,Z 329.338,A -85,B 0,C 180,E1 -18596.646,E2 -18596.646} C_VEL
LIN {X 0,Y 168.995,Z 312.844,A -85,B 0,C 180,E1 -18595.934,E2 -18595.934} C_VEL
LIN {X 0,Y 175.084,Z 249.207,A -85,B 0,C 180,E1 -18593.886,E2 -18593.886} C_VEL
LIN {X 0,Y 171.673,Z 241.39,A -85,B 0,C 180,E1 -18591.651,E2 -18591.651} C_VEL
LIN {X 0,Y 168.74,Z 248.446,A -85,B 0,C 180,E1 -18590.723,E2 -18590.723} C_VEL
LIN {X 0,Y 167.013,Z 252.1,A -85,B 0,C 180,E1 -18590.107,E2 -18590.107} C_VEL
LIN {X 0,Y 160.891,Z 274.728,A -85,B 0,C 180,E1 -18588.659,E2 -18588.659} C_VEL
LIN {X 0,Y 156.181,Z 289.747,A -85,B 0,C 180,E1 -18587.228,E2 -18587.228} C_VEL
LIN {X 0,Y 152.818,Z 298.829,A -85,B 0,C 180,E1 -18585.939,E2 -18585.939} C_VEL
LIN {X 0,Y 150.211,Z 304.359,A -85,B 0,C 180,E1 -18584.692,E2 -18584.692} C_VEL
LIN {X 0,Y 146.107,Z 318.482,A -85,B 0,C 180,E1 -18583.361,E2 -18583.361} C_VEL
LIN {X 0,Y 141.933,Z 329.242,A -85,B 0,C 180,E1 -18581.945,E2 -18581.945} C_VEL
LIN {X 0,Y 137.939,Z 337.219,A -85,B 0,C 180,E1 -18580.394,E2 -18580.394} C_VEL
LIN {X 0,Y 134.526,Z 342.804,A -85,B 0,C 180,E1 -18578.824,E2 -18578.824} C_VEL
LIN {X 0,Y 130.419,Z 347.972,A -85,B 0,C 180,E1 -18576.355,E2 -18576.355} C_VEL
LIN {X 0,Y 126.566,Z 354.423,A -85,B 0,C 180,E1 -18574.694,E2 -18574.694} C_VEL
LIN {X 0,Y 123.099,Z 359.414,A -85,B 0,C 180,E1 -18572.847,E2 -18572.847} C_VEL
LIN {X 0,Y 121.159,Z 361.822,A -85,B 0,C 180,E1 -18571.472,E2 -18571.472} C_VEL
LIN {X 0,Y 117.972,Z 365.013,A -85,B 0,C 180,E1 -18568.464,E2 -18568.464} C_VEL
LIN {X 0,Y 114.726,Z 369.752,A -85,B 0,C 180,E1 -18566.369,E2 -18566.369} C_VEL
LIN {X 0,Y 112.134,Z 373.143,A -85,B 0,C 180,E1 -18564.042,E2 -18564.042} C_VEL
LIN {X 0,Y 110.857,Z 374.624,A -85,B 0,C 180,E1 -18562.359,E2 -18562.359} C_VEL
LIN {X 0,Y 110.27,Z 375.08,A -85,B 0,C 180,E1 -18560.4,E2 -18560.4} C_VEL
LIN {X 0,Y 108.702,Z 387.123,A -85,B 0,C 180,E1 -18554.989,E2 -18554.989} C_VEL
LIN {X 0,Y 107.631,Z 398.536,A -85,B 0,C 180,E1 -18548.815,E2 -18548.815} C_VEL
LIN {X 0,Y 107.29,Z 406.479,A -85,B 0,C 180,E1 -18543.757,E2 -18543.757} C_VEL
LIN {X 0,Y 107.444,Z 415.121,A -85,B 0,C 180,E1 -18537.189,E2 -18537.189} C_VEL
LIN {X 0,Y 108.06,Z 422.33,A -85,B 0,C 180,E1 -18530.644,E2 -18530.644} C_VEL
LIN {X 0,Y 110.807,Z 430.738,A -85,B 0,C 180,E1 -18521.512,E2 -18521.512} C_VEL
LIN {X 0,Y 116.123,Z 437.472,A -85,B 0,C 180,E1 -18513.006,E2 -18513.006} C_VEL
LIN {X 0,Y 123.86,Z 442.828,A -85,B 0,C 180,E1 -18505.431,E2 -18505.431} C_VEL
LIN {X 0,Y 131.74,Z 446.193,A -85,B 0,C 180,E1 -18500.197,E2 -18500.197} C_VEL
LIN {X 0,Y 136.228,Z 447.646,A -85,B 0,C 180,E1 -18497.882,E2 -18497.882} C_VEL
LIN {X 0,Y 136.54,Z 447.887,A -85,B 0,C 180,E1 -18496.915,E2 -18496.915} C_VEL
LIN {X 0,Y 127.188,Z 446.595,A -85,B 0,C 180,E1 -18491.535,E2 -18491.535} C_VEL
LIN {X 0,Y 118.205,Z 444.08,A -85,B 0,C 180,E1 -18484.004,E2 -18484.004} C_VEL
LIN {X 0,Y 113.475,Z 449.514,A -85,B 0,C 180,E1 -18479.701,E2 -18479.701} C_VEL
LIN {X 0,Y 108.839,Z 455.991,A -85,B 0,C 180,E1 -18472.795,E2 -18472.795} C_VEL
LIN {X 0,Y 106.163,Z 460.998,A -85,B 0,C 180,E1 -18465.355,E2 -18465.355} C_VEL
LIN {X 0,Y 105.117,Z 464.628,A -85,B 0,C 180,E1 -18457.684,E2 -18457.684} C_VEL
LIN {X 0,Y 105.076,Z 465.949,A -85,B 0,C 180,E1 -18453.835,E2 -18453.835} C_VEL
LIN {X 0,Y 105.171,Z 466.949,A -85,B 0,C 180,E1 -18450,E2 -18450} C_VEL
LIN {X 0,Y 105.129,Z 468.012,A -85,B 0,C 180,E1 -18442.316,E2 -18442.316} C_VEL
LIN {X 0,Y 106.234,Z 467.902,A -85,B 0,C 180,E1 -18434.655,E2 -18434.655} C_VEL
LIN {X 0,Y 108.997,Z 466.665,A -85,B 0,C 180,E1 -18427.24,E2 -18427.24} C_VEL
LIN {X 0,Y 113.41,Z 464.285,A -85,B 0,C 180,E1 -18420.177,E2 -18420.177} C_VEL
LIN {X 0,Y 119.422,Z 460.836,A -85,B 0,C 180,E1 -18413.949,E2 -18413.949} C_VEL
LIN {X 0,Y 126.873,Z 456.124,A -85,B 0,C 180,E1 -18408.339,E2 -18408.339} C_VEL
LIN {X 0,Y 135.65,Z 450.039,A -85,B 0,C 180,E1 -18403.503,E2 -18403.503} C_VEL
LIN {X 0,Y 136.522,Z 449.401,A -85,B 0,C 180,E1 -18403.123,E2 -18403.123} C_VEL
LIN {X 0,Y 136.117,Z 448.878,A -85,B 0,C 180,E1 -18402.16,E2 -18402.16} C_VEL
LIN {X 0,Y 128.049,Z 449.208,A -85,B 0,C 180,E1 -18397.137,E2 -18397.137} C_VEL
LIN {X 0,Y 116.001,Z 449.654,A -85,B 0,C 180,E1 -18384.662,E2 -18384.662} C_VEL
LIN {X 0,Y 111.513,Z 450.285,A -85,B 0,C 180,E1 -18363.612,E2 -18363.612} C_VEL
LIN {X 0,Y 116.094,Z 451.512,A -85,B 0,C 180,E1 -18349.535,E2 -18349.535} C_VEL
LIN {X 0,Y 125.815,Z 453.287,A -85,B 0,C 180,E1 -18336.981,E2 -18336.981} C_VEL
LIN {X 0,Y 124.015,Z 454.678,A -85,B 0,C 180,E1 -18335.057,E2 -18335.057} C_VEL
LIN {X 0,Y 119.896,Z 457.111,A -85,B 0,C 180,E1 -18331.554,E2 -18331.554} C_VEL
LIN {X 0,Y 115.289,Z 459.543,A -85,B 0,C 180,E1 -18326.725,E2 -18326.725} C_VEL
LIN {X 0,Y 110.417,Z 461.778,A -85,B 0,C 180,E1 -18319.8,E2 -18319.8} C_VEL
LIN {X 0,Y 106.605,Z 462.891,A -85,B 0,C 180,E1 -18311.243,E2 -18311.243} C_VEL
LIN {X 0,Y 104.972,Z 462.664,A -85,B 0,C 180,E1 -18304.422,E2 -18304.422} C_VEL
LIN {X 0,Y 104.363,Z 462.475,A -85,B 0,C 180,E1 -18302.3,E2 -18302.3} C_VEL
LIN {X 0,Y 102.1,Z 461.817,A -85,B 0,C 180,E1 -18298.115,E2 -18298.115} C_VEL
LIN {X 0,Y 98.593,Z 460.098,A -85,B 0,C 180,E1 -18291.644,E2 -18291.644} C_VEL
LIN {X 0,Y 98.022,Z 458.904,A -85,B 0,C 180,E1 -18288.25,E2 -18288.25} C_VEL
LIN {X 0,Y 98.156,Z 458.426,A -85,B 0,C 180,E1 -18287.116,E2 -18287.116} C_VEL
LIN {X 0,Y 99.998,Z 455.141,A -85,B 0,C 180,E1 -18280.276,E2 -18280.276} C_VEL
LIN {X 0,Y 102.577,Z 451.053,A -85,B 0,C 180,E1 -18273.929,E2 -18273.929} C_VEL
LIN {X 0,Y 107.315,Z 444.36,A -85,B 0,C 180,E1 -18266.245,E2 -18266.245} C_VEL
LIN {X 0,Y 112.684,Z 437.068,A -85,B 0,C 180,E1 -18260.124,E2 -18260.124} C_VEL
LIN {X 0,Y 119.121,Z 428.205,A -85,B 0,C 180,E1 -18254.604,E2 -18254.604} C_VEL
LIN {X 0,Y 126.194,Z 417.772,A -85,B 0,C 180,E1 -18249.772,E2 -18249.772} C_VEL
LIN {X 0,Y 133.255,Z 406.422,A -85,B 0,C 180,E1 -18245.874,E2 -18245.874} C_VEL
LIN {X 0,Y 139.943,Z 394.299,A -85,B 0,C 180,E1 -18242.725,E2 -18242.725} C_VEL
LIN {X 0,Y 146.041,Z 381.66,A -85,B 0,C 180,E1 -18240.231,E2 -18240.231} C_VEL
LIN {X 0,Y 151.598,Z 368.061,A -85,B 0,C 180,E1 -18238.174,E2 -18238.174} C_VEL
LIN {X 0,Y 156.644,Z 352.987,A -85,B 0,C 180,E1 -18236.467,E2 -18236.467} C_VEL
LIN {X 0,Y 160.358,Z 338.647,A -85,B 0,C 180,E1 -18235.267,E2 -18235.267} C_VEL
LIN {X 0,Y 163.295,Z 323.357,A -85,B 0,C 180,E1 -18234.381,E2 -18234.381} C_VEL
LIN {X 0,Y 165.752,Z 302.91,A -85,B 0,C 180,E1 -18233.671,E2 -18233.671} C_VEL
LIN {X 0,Y 170.493,Z 255.333,A -85,B 0,C 180,E1 -18232.187,E2 -18232.187} C_VEL
LIN {X 0,Y 170.458,Z 254.549,A -85,B 0,C 180,E1 -18232.107,E2 -18232.107} C_VEL
LIN {X 0,Y 163.715,Z 278.526,A -85,B 0,C 180,E1 -18230.599,E2 -18230.599} C_VEL
LIN {X 0,Y 159.254,Z 292.442,A -85,B 0,C 180,E1 -18229.333,E2 -18229.333} C_VEL
LIN {X 0,Y 155.601,Z 301.998,A -85,B 0,C 180,E1 -18228.061,E2 -18228.061} C_VEL
LIN {X 0,Y 152.847,Z 307.782,A -85,B 0,C 180,E1 -18226.883,E2 -18226.883} C_VEL
LIN {X 0,Y 148.612,Z 321.456,A -85,B 0,C 180,E1 -18225.667,E2 -18225.667} C_VEL
LIN {X 0,Y 144.015,Z 332.536,A -85,B 0,C 180,E1 -18224.319,E2 -18224.319} C_VEL
LIN {X 0,Y 139.708,Z 340.517,A -85,B 0,C 180,E1 -18222.899,E2 -18222.899} C_VEL
LIN {X 0,Y 135.712,Z 346.691,A -85,B 0,C 180,E1 -18221.322,E2 -18221.322} C_VEL
LIN {X 0,Y 132.298,Z 350.813,A -85,B 0,C 180,E1 -18219.605,E2 -18219.605} C_VEL
LIN {X 0,Y 131.232,Z 352.001,A -85,B 0,C 180,E1 -18218.997,E2 -18218.997} C_VEL
LIN {X 0,Y 125.881,Z 359.89,A -85,B 0,C 180,E1 -18216.884,E2 -18216.884} C_VEL
LIN {X 0,Y 122.233,Z 364.535,A -85,B 0,C 180,E1 -18215.099,E2 -18215.099} C_VEL
LIN {X 0,Y 120.126,Z 366.92,A -85,B 0,C 180,E1 -18213.767,E2 -18213.767} C_VEL
LIN {X 0,Y 116.564,Z 370.268,A -85,B 0,C 180,E1 -18210.831,E2 -18210.831} C_VEL
LIN {X 0,Y 113.114,Z 374.716,A -85,B 0,C 180,E1 -18208.786,E2 -18208.786} C_VEL
LIN {X 0,Y 110.225,Z 378.027,A -85,B 0,C 180,E1 -18206.509,E2 -18206.509} C_VEL
LIN {X 0,Y 108.719,Z 379.617,A -85,B 0,C 180,E1 -18204.848,E2 -18204.848} C_VEL
LIN {X 0,Y 106.908,Z 381.37,A -85,B 0,C 180,E1 -18202.109,E2 -18202.109} C_VEL
LIN {X 0,Y 104.327,Z 384.715,A -85,B 0,C 180,E1 -18199.685,E2 -18199.685} C_VEL
LIN {X 0,Y 102.907,Z 386.58,A -85,B 0,C 180,E1 -18197.9,E2 -18197.9} C_VEL
LIN {X 0,Y 101.914,Z 387.934,A -85,B 0,C 180,E1 -18196.013,E2 -18196.013} C_VEL
LIN {X 0,Y 101.421,Z 388.658,A -85,B 0,C 180,E1 -18193.571,E2 -18193.571} C_VEL
LIN {X 0,Y 101.488,Z 388.632,A -85,B 0,C 180,E1 -18193.087,E2 -18193.087} C_VEL
LIN {X 0,Y 100.786,Z 397.363,A -85,B 0,C 180,E1 -18188.018,E2 -18188.018} C_VEL
LIN {X 0,Y 100.561,Z 407.508,A -85,B 0,C 180,E1 -18181.002,E2 -18181.002} C_VEL
LIN {X 0,Y 100.856,Z 414.79,A -85,B 0,C 180,E1 -18175.004,E2 -18175.004} C_VEL
LIN {X 0,Y 101.427,Z 419.975,A -85,B 0,C 180,E1 -18170.026,E2 -18170.026} C_VEL
LIN {X 0,Y 104.009,Z 428.145,A -85,B 0,C 180,E1 -18161.084,E2 -18161.084} C_VEL
LIN {X 0,Y 108.675,Z 434.637,A -85,B 0,C 180,E1 -18153.085,E2 -18153.085} C_VEL
LIN {X 0,Y 116.33,Z 440.624,A -85,B 0,C 180,E1 -18144.976,E2 -18144.976} C_VEL
LIN {X 0,Y 127.369,Z 445.725,A -85,B 0,C 180,E1 -18137.65,E2 -18137.65} C_VEL
LIN {X 0,Y 126.347,Z 445.677,A -85,B 0,C 180,E1 -18136.313,E2 -18136.313} C_VEL
LIN {X 0,Y 114.545,Z 442.732,A -85,B 0,C 180,E1 -18127.847,E2 -18127.847} C_VEL
LIN {X 0,Y 113.317,Z 442.297,A -85,B 0,C 180,E1 -18126.652,E2 -18126.652} C_VEL
LIN {X 0,Y 107.369,Z 448.793,A -85,B 0,C 180,E1 -18121.578,E2 -18121.578} C_VEL
LIN {X 0,Y 102.266,Z 455.373,A -85,B 0,C 180,E1 -18114.352,E2 -18114.352} C_VEL
LIN {X 0,Y 99.258,Z 460.485,A -85,B 0,C 180,E1 -18106.453,E2 -18106.453} C_VEL
LIN {X 0,Y 98.052,Z 464.219,A -85,B 0,C 180,E1 -18098.242,E2 -18098.242} C_VEL
LIN {X 0,Y 97.987,Z 465.59,A -85,B 0,C 180,E1 -18094.113,E2 -18094.113} C_VEL
LIN {X 0,Y 98.074,Z 466.638,A -85,B 0,C 180,E1 -18090,E2 -18090} C_VEL
LIN {X 0,Y 98.066,Z 467.778,A -85,B 0,C 180,E1 -18081.759,E2 -18081.759} C_VEL
LIN {X 0,Y 99.337,Z 467.738,A -85,B 0,C 180,E1 -18073.561,E2 -18073.561} C_VEL
LIN {X 0,Y 102.418,Z 466.604,A -85,B 0,C 180,E1 -18065.687,E2 -18065.687} C_VEL
LIN {X 0,Y 107.203,Z 464.378,A -85,B 0,C 180,E1 -18058.368,E2 -18058.368} C_VEL
LIN {X 0,Y 113.724,Z 461.013,A -85,B 0,C 180,E1 -18051.831,E2 -18051.831} C_VEL
LIN {X 0,Y 121.647,Z 456.418,A -85,B 0,C 180,E1 -18046.109,E2 -18046.109} C_VEL
LIN {X 0,Y 127.884,Z 452.442,A -85,B 0,C 180,E1 -18042.7,E2 -18042.7} C_VEL
LIN {X 0,Y 126.959,Z 452.162,A -85,B 0,C 180,E1 -18041.626,E2 -18041.626} C_VEL
LIN {X 0,Y 112.982,Z 452.469,A -85,B 0,C 180,E1 -18029.843,E2 -18029.843} C_VEL
LIN {X 0,Y 104.926,Z 453.02,A -85,B 0,C 180,E1 -18003.839,E2 -18003.839} C_VEL
LIN {X 0,Y 109.568,Z 454.04,A -85,B 0,C 180,E1 -17988.904,E2 -17988.904} C_VEL
LIN {X 0,Y 117.904,Z 455.357,A -85,B 0,C 180,E1 -17977.365,E2 -17977.365} C_VEL
LIN {X 0,Y 115.522,Z 456.871,A -85,B 0,C 180,E1 -17974.794,E2 -17974.794} C_VEL
LIN {X 0,Y 108.278,Z 460.383,A -85,B 0,C 180,E1 -17967.543,E2 -17967.543} C_VEL
LIN {X 0,Y 104.863,Z 461.784,A -85,B 0,C 180,E1 -17962.9,E2 -17962.9} C_VEL
LIN {X 0,Y 100.5,Z 463.044,A -85,B 0,C 180,E1 -17954.371,E2 -17954.371} C_VEL
LIN {X 0,Y 98.654,Z 463.08,A -85,B 0,C 180,E1 -17948.404,E2 -17948.404} C_VEL
LIN {X 0,Y 97.396,Z 462.178,A -85,B 0,C 180,E1 -17940.011,E2 -17940.011} C_VEL
LIN {X 0,Y 97.572,Z 459.923,A -85,B 0,C 180,E1 -17931.109,E2 -17931.109} C_VEL
LIN {X 0,Y 98.156,Z 458.426,A -85,B 0,C 180,E1 -17927.116,E2 -17927.116} C_VEL
LIN {X 0,Y 98.261,Z 457.05,A -85,B 0,C 180,E1 -17923.767,E2 -17923.767} C_VEL
LIN {X 0,Y 97.093,Z 454.353,A -85,B 0,C 180,E1 -17918.204,E2 -17918.204} C_VEL
LIN {X 0,Y 96.474,Z 451.762,A -85,B 0,C 180,E1 -17913.73,E2 -17913.73} C_VEL
LIN {X 0,Y 97.07,Z 449.514,A -85,B 0,C 180,E1 -17910.478,E2 -17910.478} C_VEL
LIN {X 0,Y 97.578,Z 448.703,A -85,B 0,C 180,E1 -17909.452,E2 -17909.452} C_VEL
LIN {X 0,Y 102.885,Z 441.857,A -85,B 0,C 180,E1 -17902.148,E2 -17902.148} C_VEL
LIN {X 0,Y 108.823,Z 434.216,A -85,B 0,C 180,E1 -17896.157,E2 -17896.157} C_VEL
LIN {X 0,Y 115.103,Z 425.933,A -85,B 0,C 180,E1 -17891.303,E2 -17891.303} C_VEL
LIN {X 0,Y 122.443,Z 415.413,A -85,B 0,C 180,E1 -17886.692,E2 -17886.692} C_VEL
LIN {X 0,Y 129.653,Z 404.025,A -85,B 0,C 180,E1 -17883.001,E2 -17883.001} C_VEL
LIN {X 0,Y 136.038,Z 392.641,A -85,B 0,C 180,E1 -17880.182,E2 -17880.182} C_VEL
LIN {X 0,Y 142.448,Z 379.459,A -85,B 0,C 180,E1 -17877.704,E2 -17877.704} C_VEL
LIN {X 0,Y 148.182,Z 365.423,A -85,B 0,C 180,E1 -17875.722,E2 -17875.722} C_VEL
LIN {X 0,Y 153.066,Z 350.636,A -85,B 0,C 180,E1 -17874.168,E2 -17874.168} C_VEL
LIN {X 0,Y 156.842,Z 335.52,A -85,B 0,C 180,E1 -17872.977,E2 -17872.977} C_VEL
LIN {X 0,Y 159.736,Z 319.653,A -85,B 0,C 180,E1 -17872.178,E2 -17872.178} C_VEL
LIN {X 0,Y 162.356,Z 296.315,A -85,B 0,C 180,E1 -17871.406,E2 -17871.406} C_VEL
LIN {X 0,Y 162.382,Z 295.396,A -85,B 0,C 180,E1 -17871.34,E2 -17871.34} C_VEL
LIN {X 0,Y 158.574,Z 305.21,A -85,B 0,C 180,E1 -17870.1,E2 -17870.1} C_VEL
LIN {X 0,Y 155.511,Z 311.872,A -85,B 0,C 180,E1 -17868.953,E2 -17868.953} C_VEL
LIN {X 0,Y 151.075,Z 324.892,A -85,B 0,C 180,E1 -17867.853,E2 -17867.853} C_VEL
LIN {X 0,Y 146.189,Z 335.809,A -85,B 0,C 180,E1 -17866.648,E2 -17866.648} C_VEL
LIN {X 0,Y 141.861,Z 343.46,A -85,B 0,C 180,E1 -17865.412,E2 -17865.412} C_VEL
LIN {X 0,Y 136.8,Z 350.77,A -85,B 0,C 180,E1 -17863.716,E2 -17863.716} C_VEL
LIN {X 0,Y 133.446,Z 354.79,A -85,B 0,C 180,E1 -17862.302,E2 -17862.302} C_VEL
LIN {X 0,Y 130.899,Z 357.597,A -85,B 0,C 180,E1 -17861.127,E2 -17861.127} C_VEL
LIN {X 0,Y 125.265,Z 365.168,A -85,B 0,C 180,E1 -17859.139,E2 -17859.139} C_VEL
LIN {X 0,Y 121.443,Z 369.565,A -85,B 0,C 180,E1 -17857.421,E2 -17857.421} C_VEL
LIN {X 0,Y 119.149,Z 371.877,A -85,B 0,C 180,E1 -17856.148,E2 -17856.148} C_VEL
LIN {X 0,Y 115.261,Z 375.339,A -85,B 0,C 180,E1 -17853.284,E2 -17853.284} C_VEL
LIN {X 0,Y 110.448,Z 380.728,A -85,B 0,C 180,E1 -17850.602,E2 -17850.602} C_VEL
LIN {X 0,Y 108.419,Z 382.791,A -85,B 0,C 180,E1 -17849.09,E2 -17849.09} C_VEL
LIN {X 0,Y 106.657,Z 384.435,A -85,B 0,C 180,E1 -17847.47,E2 -17847.47} C_VEL
LIN {X 0,Y 103.683,Z 387.226,A -85,B 0,C 180,E1 -17843.999,E2 -17843.999} C_VEL
LIN {X 0,Y 100.161,Z 391.19,A -85,B 0,C 180,E1 -17840.54,E2 -17840.54} C_VEL
LIN {X 0,Y 98.875,Z 392.633,A -85,B 0,C 180,E1 -17838.656,E2 -17838.656} C_VEL
LIN {X 0,Y 97.951,Z 393.715,A -85,B 0,C 180,E1 -17836.68,E2 -17836.68} C_VEL
LIN {X 0,Y 97.399,Z 394.429,A -85,B 0,C 180,E1 -17834.64,E2 -17834.64} C_VEL
LIN {X 0,Y 94.828,Z 398.066,A -85,B 0,C 180,E1 -17830.679,E2 -17830.679} C_VEL
LIN {X 0,Y 94.02,Z 399.466,A -85,B 0,C 180,E1 -17828.599,E2 -17828.599} C_VEL
LIN {X 0,Y 93.718,Z 401.288,A -85,B 0,C 180,E1 -17823.764,E2 -17823.764} C_VEL
LIN {X 0,Y 93.844,Z 401.531,A -85,B 0,C 180,E1 -17823.221,E2 -17823.221} C_VEL
LIN {X 0,Y 94.063,Z 409.619,A -85,B 0,C 180,E1 -17816.789,E2 -17816.789} C_VEL
LIN {X 0,Y 94.853,Z 417.496,A -85,B 0,C 180,E1 -17809.327,E2 -17809.327} C_VEL
LIN {X 0,Y 98.006,Z 426.709,A -85,B 0,C 180,E1 -17798.99,E2 -17798.99} C_VEL
LIN {X 0,Y 104.042,Z 434.189,A -85,B 0,C 180,E1 -17789.562,E2 -17789.562} C_VEL
LIN {X 0,Y 112.676,Z 440.253,A -85,B 0,C 180,E1 -17781.412,E2 -17781.412} C_VEL
LIN {X 0,Y 118.078,Z 442.936,A -85,B 0,C 180,E1 -17777.769,E2 -17777.769} C_VEL
LIN {X 0,Y 117.225,Z 442.941,A -85,B 0,C 180,E1 -17776.008,E2 -17776.008} C_VEL
LIN {X 0,Y 108.675,Z 440.457,A -85,B 0,C 180,E1 -17769.539,E2 -17769.539} C_VEL
LIN {X 0,Y 101.754,Z 447.676,A -85,B 0,C 180,E1 -17764.024,E2 -17764.024} C_VEL
LIN {X 0,Y 96.992,Z 453.192,A -85,B 0,C 180,E1 -17758.098,E2 -17758.098} C_VEL
LIN {X 0,Y 93.084,Z 458.776,A -85,B 0,C 180,E1 -17749.862,E2 -17749.862} C_VEL
LIN {X 0,Y 91.496,Z 462.049,A -85,B 0,C 180,E1 -17743.323,E2 -17743.323} C_VEL
LIN {X 0,Y 90.892,Z 465.226,A -85,B 0,C 180,E1 -17734.435,E2 -17734.435} C_VEL
LIN {X 0,Y 90.972,Z 466.316,A -85,B 0,C 180,E1 -17730,E2 -17730} C_VEL
LIN {X 0,Y 91.027,Z 467.515,A -85,B 0,C 180,E1 -17721.117,E2 -17721.117} C_VEL
LIN {X 0,Y 92.486,Z 467.576,A -85,B 0,C 180,E1 -17712.304,E2 -17712.304} C_VEL
LIN {X 0,Y 95.927,Z 466.553,A -85,B 0,C 180,E1 -17703.923,E2 -17703.923} C_VEL
LIN {X 0,Y 101.19,Z 464.44,A -85,B 0,C 180,E1 -17696.246,E2 -17696.246} C_VEL
LIN {X 0,Y 108.207,Z 461.177,A -85,B 0,C 180,E1 -17689.497,E2 -17689.497} C_VEL
LIN {X 0,Y 116.623,Z 456.685,A -85,B 0,C 180,E1 -17683.685,E2 -17683.685} C_VEL
LIN {X 0,Y 118.2,Z 455.803,A -85,B 0,C 180,E1 -17682.814,E2 -17682.814} C_VEL
LIN {X 0,Y 118.825,Z 454.984,A -85,B 0,C 180,E1 -17681.553,E2 -17681.553} C_VEL
LIN {X 0,Y 104.518,Z 455.217,A -85,B 0,C 180,E1 -17668.078,E2 -17668.078} C_VEL
LIN {X 0,Y 98.766,Z 455.665,A -85,B 0,C 180,E1 -17639.999,E2 -17639.999} C_VEL
LIN {X 0,Y 102.964,Z 456.31,A -85,B 0,C 180,E1 -17628.183,E2 -17628.183} C_VEL
LIN {X 0,Y 110.208,Z 457.232,A -85,B 0,C 180,E1 -17617.503,E2 -17617.503} C_VEL
LIN {X 0,Y 103.962,Z 460.082,A -85,B 0,C 180,E1 -17611.501,E2 -17611.501} C_VEL
LIN {X 0,Y 97.2,Z 462.488,A -85,B 0,C 180,E1 -17602.688,E2 -17602.688} C_VEL
LIN {X 0,Y 92.756,Z 463.328,A -85,B 0,C 180,E1 -17592.994,E2 -17592.994} C_VEL
LIN {X 0,Y 91.384,Z 463.181,A -85,B 0,C 180,E1 -17587.97,E2 -17587.97} C_VEL
LIN {X 0,Y 90.357,Z 462.408,A -85,B 0,C 180,E1 -17581.173,E2 -17581.173} C_VEL
LIN {X 0,Y 90.463,Z 460.065,A -85,B 0,C 180,E1 -17571.205,E2 -17571.205} C_VEL
LIN {X 0,Y 91.919,Z 457.086,A -85,B 0,C 180,E1 -17563.26,E2 -17563.26} C_VEL
LIN {X 0,Y 94.14,Z 453.5,A -85,B 0,C 180,E1 -17556.43,E2 -17556.43} C_VEL
LIN {X 0,Y 97.578,Z 448.703,A -85,B 0,C 180,E1 -17549.452,E2 -17549.452} C_VEL
LIN {X 0,Y 98.82,Z 446.288,A -85,B 0,C 180,E1 -17546.403,E2 -17546.403} C_VEL
LIN {X 0,Y 99.651,Z 441.952,A -85,B 0,C 180,E1 -17541.246,E2 -17541.246} C_VEL
LIN {X 0,Y 101.099,Z 437.204,A -85,B 0,C 180,E1 -17536.332,E2 -17536.332} C_VEL
LIN {X 0,Y 103.195,Z 433.978,A -85,B 0,C 180,E1 -17533.812,E2 -17533.812} C_VEL
LIN {X 0,Y 110.339,Z 424.949,A -85,B 0,C 180,E1 -17528.516,E2 -17528.516} C_VEL
LIN {X 0,Y 117.928,Z 414.534,A -85,B 0,C 180,E1 -17524.043,E2 -17524.043} C_VEL
LIN {X 0,Y 125.052,Z 403.619,A -85,B 0,C 180,E1 -17520.544,E2 -17520.544} C_VEL
LIN {X 0,Y 131.707,Z 392.116,A -85,B 0,C 180,E1 -17517.75,E2 -17517.75} C_VEL
LIN {X 0,Y 137.932,Z 379.765,A -85,B 0,C 180,E1 -17515.469,E2 -17515.469} C_VEL
LIN {X 0,Y 143.6,Z 366.456,A -85,B 0,C 180,E1 -17513.6,E2 -17513.6} C_VEL
LIN {X 0,Y 148.627,Z 351.902,A -85,B 0,C 180,E1 -17512.068,E2 -17512.068} C_VEL
LIN {X 0,Y 152.65,Z 336.571,A -85,B 0,C 180,E1 -17510.864,E2 -17510.864} C_VEL
LIN {X 0,Y 154.783,Z 326.174,A -85,B 0,C 180,E1 -17510.303,E2 -17510.303} C_VEL
LIN {X 0,Y 154.633,Z 326.046,A -85,B 0,C 180,E1 -17510.198,E2 -17510.198} C_VEL
LIN {X 0,Y 149.605,Z 337.03,A -85,B 0,C 180,E1 -17509.148,E2 -17509.148} C_VEL
LIN {X 0,Y 144.224,Z 346.358,A -85,B 0,C 180,E1 -17507.87,E2 -17507.87} C_VEL
LIN {X 0,Y 138.262,Z 354.61,A -85,B 0,C 180,E1 -17506.152,E2 -17506.152} C_VEL
LIN {X 0,Y 133.39,Z 360.027,A -85,B 0,C 180,E1 -17504.357,E2 -17504.357} C_VEL
LIN {X 0,Y 132.051,Z 361.334,A -85,B 0,C 180,E1 -17503.781,E2 -17503.781} C_VEL
LIN {X 0,Y 124.742,Z 370.273,A -85,B 0,C 180,E1 -17501.454,E2 -17501.454} C_VEL
LIN {X 0,Y 119.497,Z 375.634,A -85,B 0,C 180,E1 -17499.217,E2 -17499.217} C_VEL
LIN {X 0,Y 116.048,Z 378.574,A -85,B 0,C 180,E1 -17497.274,E2 -17497.274} C_VEL
LIN {X 0,Y 113.986,Z 380.212,A -85,B 0,C 180,E1 -17495.856,E2 -17495.856} C_VEL
LIN {X 0,Y 109.134,Z 385.179,A -85,B 0,C 180,E1 -17493.41,E2 -17493.41} C_VEL
LIN {X 0,Y 106.689,Z 387.452,A -85,B 0,C 180,E1 -17491.804,E2 -17491.804} C_VEL
LIN {X 0,Y 102.996,Z 390.479,A -85,B 0,C 180,E1 -17488.534,E2 -17488.534} C_VEL
LIN {X 0,Y 101.361,Z 391.839,A -85,B 0,C 180,E1 -17486.789,E2 -17486.789} C_VEL
LIN {X 0,Y 97.533,Z 395.682,A -85,B 0,C 180,E1 -17483.35,E2 -17483.35} C_VEL
LIN {X 0,Y 94.713,Z 398.382,A -85,B 0,C 180,E1 -17479.508,E2 -17479.508} C_VEL
LIN {X 0,Y 93.785,Z 399.319,A -85,B 0,C 180,E1 -17477.444,E2 -17477.444} C_VEL
LIN {X 0,Y 90.149,Z 403.857,A -85,B 0,C 180,E1 -17471.24,E2 -17471.24} C_VEL
LIN {X 0,Y 89.465,Z 404.963,A -85,B 0,C 180,E1 -17469.041,E2 -17469.041} C_VEL
LIN {X 0,Y 88.996,Z 406.608,A -85,B 0,C 180,E1 -17464.531,E2 -17464.531} C_VEL
LIN {X 0,Y 87.559,Z 409.742,A -85,B 0,C 180,E1 -17460.001,E2 -17460.001} C_VEL
LIN {X 0,Y 87.273,Z 413.419,A -85,B 0,C 180,E1 -17453.064,E2 -17453.064} C_VEL
LIN {X 0,Y 88.566,Z 415.794,A -85,B 0,C 180,E1 -17447.397,E2 -17447.397} C_VEL
LIN {X 0,Y 91.765,Z 424.386,A -85,B 0,C 180,E1 -17437.486,E2 -17437.486} C_VEL
LIN {X 0,Y 98.223,Z 432.261,A -85,B 0,C 180,E1 -17427.546,E2 -17427.546} C_VEL
LIN {X 0,Y 108.984,Z 439.578,A -85,B 0,C 180,E1 -17417.942,E2 -17417.942} C_VEL
LIN {X 0,Y 109.313,Z 439.958,A -85,B 0,C 180,E1 -17416.363,E2 -17416.363} C_VEL
LIN {X 0,Y 104.395,Z 438.534,A -85,B 0,C 180,E1 -17412.642,E2 -17412.642} C_VEL
LIN {X 0,Y 97.493,Z 445.284,A -85,B 0,C 180,E1 -17407.788,E2 -17407.788} C_VEL
LIN {X 0,Y 92.208,Z 450.878,A -85,B 0,C 180,E1 -17402.245,E2 -17402.245} C_VEL
LIN {X 0,Y 87.271,Z 456.944,A -85,B 0,C 180,E1 -17393.744,E2 -17393.744} C_VEL
LIN {X 0,Y 84.55,Z 461.571,A -85,B 0,C 180,E1 -17384.44,E2 -17384.44} C_VEL
LIN {X 0,Y 83.79,Z 464.825,A -85,B 0,C 180,E1 -17374.811,E2 -17374.811} C_VEL
LIN {X 0,Y 83.897,Z 465.953,A -85,B 0,C 180,E1 -17370,E2 -17370} C_VEL
LIN {X 0,Y 83.985,Z 467.246,A -85,B 0,C 180,E1 -17360.365,E2 -17360.365} C_VEL
LIN {X 0,Y 85.688,Z 467.415,A -85,B 0,C 180,E1 -17350.848,E2 -17350.848} C_VEL
LIN {X 0,Y 89.541,Z 466.503,A -85,B 0,C 180,E1 -17341.905,E2 -17341.905} C_VEL
LIN {X 0,Y 95.329,Z 464.497,A -85,B 0,C 180,E1 -17333.858,E2 -17333.858} C_VEL
LIN {X 0,Y 102.897,Z 461.323,A -85,B 0,C 180,E1 -17326.921,E2 -17326.921} C_VEL
LIN {X 0,Y 109.093,Z 458.402,A -85,B 0,C 180,E1 -17322.698,E2 -17322.698} C_VEL
LIN {X 0,Y 109.88,Z 457.516,A -85,B 0,C 180,E1 -17321.028,E2 -17321.028} C_VEL
LIN {X 0,Y 94.131,Z 457.62,A -85,B 0,C 180,E1 -17301.918,E2 -17301.918} C_VEL
LIN {X 0,Y 91.966,Z 457.818,A -85,B 0,C 180,E1 -17279.999,E2 -17279.999} C_VEL
LIN {X 0,Y 96.304,Z 458.316,A -85,B 0,C 180,E1 -17267.352,E2 -17267.352} C_VEL
LIN {X 0,Y 102.102,Z 458.876,A -85,B 0,C 180,E1 -17258.088,E2 -17258.088} C_VEL
LIN {X 0,Y 99.136,Z 460.173,A -85,B 0,C 180,E1 -17254.825,E2 -17254.825} C_VEL
LIN {X 0,Y 92.32,Z 462.425,A -85,B 0,C 180,E1 -17246.866,E2 -17246.866} C_VEL
LIN {X 0,Y 86.818,Z 463.488,A -85,B 0,C 180,E1 -17236.766,E2 -17236.766} C_VEL
LIN {X 0,Y 85.039,Z 463.449,A -85,B 0,C 180,E1 -17231.388,E2 -17231.388} C_VEL
LIN {X 0,Y 83.374,Z 462.632,A -85,B 0,C 180,E1 -17222.544,E2 -17222.544} C_VEL
LIN {X 0,Y 83.276,Z 460.342,A -85,B 0,C 180,E1 -17211.82,E2 -17211.82} C_VEL
LIN {X 0,Y 84.427,Z 457.871,A -85,B 0,C 180,E1 -17204.462,E2 -17204.462} C_VEL
LIN {X 0,Y 86.654,Z 454.492,A -85,B 0,C 180,E1 -17196.988,E2 -17196.988} C_VEL
LIN {X 0,Y 90.937,Z 448.811,A -85,B 0,C 180,E1 -17187.953,E2 -17187.953} C_VEL
LIN {X 0,Y 96.346,Z 442.28,A -85,B 0,C 180,E1 -17180.553,E2 -17180.553} C_VEL
LIN {X 0,Y 103.195,Z 433.978,A -85,B 0,C 180,E1 -17173.812,E2 -17173.812} C_VEL
LIN {X 0,Y 105.403,Z 430.659,A -85,B 0,C 180,E1 -17171.443,E2 -17171.443} C_VEL
LIN {X 0,Y 107.757,Z 424.878,A -85,B 0,C 180,E1 -17167.267,E2 -17167.267} C_VEL
LIN {X 0,Y 110.374,Z 418.749,A -85,B 0,C 180,E1 -17163.397,E2 -17163.397} C_VEL
LIN {X 0,Y 112.858,Z 414.711,A -85,B 0,C 180,E1 -17161.582,E2 -17161.582} C_VEL
LIN {X 0,Y 120.708,Z 403.124,A -85,B 0,C 180,E1 -17157.908,E2 -17157.908} C_VEL
LIN {X 0,Y 128.08,Z 390.685,A -85,B 0,C 180,E1 -17155.005,E2 -17155.005} C_VEL
LIN {X 0,Y 134.829,Z 377.386,A -85,B 0,C 180,E1 -17152.702,E2 -17152.702} C_VEL
LIN {X 0,Y 140.482,Z 364.035,A -85,B 0,C 180,E1 -17150.965,E2 -17150.965} C_VEL
LIN {X 0,Y 144.015,Z 354.104,A -85,B 0,C 180,E1 -17149.944,E2 -17149.944} C_VEL
LIN {X 0,Y 143.644,Z 353.554,A -85,B 0,C 180,E1 -17149.537,E2 -17149.537} C_VEL
LIN {X 0,Y 138.879,Z 359.469,A -85,B 0,C 180,E1 -17148.283,E2 -17148.283} C_VEL
LIN {X 0,Y 131.936,Z 366.618,A -85,B 0,C 180,E1 -17145.981,E2 -17145.981} C_VEL
LIN {X 0,Y 125.788,Z 373.662,A -85,B 0,C 180,E1 -17144.3,E2 -17144.3} C_VEL
LIN {X 0,Y 120.107,Z 379.249,A -85,B 0,C 180,E1 -17142.294,E2 -17142.294} C_VEL
LIN {X 0,Y 115.098,Z 383.322,A -85,B 0,C 180,E1 -17139.878,E2 -17139.878} C_VEL
LIN {X 0,Y 112.841,Z 384.941,A -85,B 0,C 180,E1 -17138.524,E2 -17138.524} C_VEL
LIN {X 0,Y 107.479,Z 389.941,A -85,B 0,C 180,E1 -17136.053,E2 -17136.053} C_VEL
LIN {X 0,Y 102.908,Z 393.663,A -85,B 0,C 180,E1 -17133.119,E2 -17133.119} C_VEL
LIN {X 0,Y 99.116,Z 396.401,A -85,B 0,C 180,E1 -17129.76,E2 -17129.76} C_VEL
LIN {X 0,Y 93.212,Z 401.562,A -85,B 0,C 180,E1 -17124.501,E2 -17124.501} C_VEL
LIN {X 0,Y 89.173,Z 405.049,A -85,B 0,C 180,E1 -17118.377,E2 -17118.377} C_VEL
LIN {X 0,Y 85.765,Z 408.814,A -85,B 0,C 180,E1 -17112.785,E2 -17112.785} C_VEL
LIN {X 0,Y 84.343,Z 411.053,A -85,B 0,C 180,E1 -17107.182,E2 -17107.182} C_VEL
LIN {X 0,Y 82.04,Z 416.303,A -85,B 0,C 180,E1 -17097.547,E2 -17097.547} C_VEL
LIN {X 0,Y 83.001,Z 420.306,A -85,B 0,C 180,E1 -17087.78,E2 -17087.78} C_VEL
LIN {X 0,Y 84.509,Z 425.564,A -85,B 0,C 180,E1 -17078.025,E2 -17078.025} C_VEL
LIN {X 0,Y 87.689,Z 428.695,A -85,B 0,C 180,E1 -17071.259,E2 -17071.259} C_VEL
LIN {X 0,Y 96.123,Z 432.946,A -85,B 0,C 180,E1 -17061.578,E2 -17061.578} C_VEL
LIN {X 0,Y 100.962,Z 436.155,A -85,B 0,C 180,E1 -17057.548,E2 -17057.548} C_VEL
LIN {X 0,Y 101.46,Z 436.511,A -85,B 0,C 180,E1 -17056.662,E2 -17056.662} C_VEL
LIN {X 0,Y 100.629,Z 436.369,A -85,B 0,C 180,E1 -17056.074,E2 -17056.074} C_VEL
LIN {X 0,Y 93.092,Z 443.436,A -85,B 0,C 180,E1 -17051.344,E2 -17051.344} C_VEL
LIN {X 0,Y 86.265,Z 450.091,A -85,B 0,C 180,E1 -17044.771,E2 -17044.771} C_VEL
LIN {X 0,Y 80.768,Z 456.284,A -85,B 0,C 180,E1 -17035.79,E2 -17035.79} C_VEL
LIN {X 0,Y 77.63,Z 461.021,A -85,B 0,C 180,E1 -17025.759,E2 -17025.759} C_VEL
LIN {X 0,Y 76.713,Z 464.389,A -85,B 0,C 180,E1 -17015.256,E2 -17015.256} C_VEL
LIN {X 0,Y 76.793,Z 465.574,A -85,B 0,C 180,E1 -17010,E2 -17010} C_VEL
LIN {X 0,Y 76.699,Z 466.421,A -85,B 0,C 180,E1 -17004.743,E2 -17004.743} C_VEL
LIN {X 0,Y 77.688,Z 467.252,A -85,B 0,C 180,E1 -16994.253,E2 -16994.253} C_VEL
LIN {X 0,Y 80.856,Z 466.992,A -85,B 0,C 180,E1 -16984.24,E2 -16984.24} C_VEL
LIN {X 0,Y 86.223,Z 465.629,A -85,B 0,C 180,E1 -16975.21,E2 -16975.21} C_VEL
LIN {X 0,Y 93.532,Z 463.136,A -85,B 0,C 180,E1 -16967.448,E2 -16967.448} C_VEL
LIN {X 0,Y 101.014,Z 460.129,A -85,B 0,C 180,E1 -16961.878,E2 -16961.878} C_VEL
LIN {X 0,Y 100.883,Z 459.718,A -85,B 0,C 180,E1 -16960.438,E2 -16960.438} C_VEL
LIN {X 0,Y 85.104,Z 459.7,A -85,B 0,C 180,E1 -16919.999,E2 -16919.999} C_VEL
LIN {X 0,Y 89.585,Z 460.044,A -85,B 0,C 180,E1 -16906.386,E2 -16906.386} C_VEL
LIN {X 0,Y 94.223,Z 460.414,A -85,B 0,C 180,E1 -16898.101,E2 -16898.101} C_VEL
LIN {X 0,Y 87.807,Z 462.403,A -85,B 0,C 180,E1 -16891.297,E2 -16891.297} C_VEL
LIN {X 0,Y 81.328,Z 463.649,A -85,B 0,C 180,E1 -16881.054,E2 -16881.054} C_VEL
LIN {X 0,Y 78.669,Z 463.677,A -85,B 0,C 180,E1 -16874.38,E2 -16874.38} C_VEL
